		// State Change Condition
		IF (CIf.Job.bolAlmReset = FALSE) THEN
			IF (me.StateMachine.intStateHistory<=cSTA_PON) THEN
				me.StateMachine.intStateNext := cSTA_PONBusy;
			ELSIF (me.intCmd=cCMD_OFF) THEN
				me.StateMachine.intStateNext := cSTA_OFFBusy;
			ELSIF (me.intCmd=cCMD_RUN) THEN
				me.StateMachine.intStateNext := cSTA_OFFBusy;
			END_IF
		END_IF
	END_IF




//--------------------------------------------------------------------------------------
// Exit action
	IF (me.StateMachine.intState<>me.StateMachine.intStateNext) THEN
		;
	END_IF
END_METHOD

METHOD PROTECTED sta_OFF : BOOL
// state implemetation
//--------------------------------------------------------------------------------------
// Entry action
	IF (me.StateMachine.intState<>me.StateMachine.intStateLastCycle) THEN
		me.StateMachine.intStateLastCycle := me.StateMachine.intState;
		
	END_IF


//--------------------------------------------------------------------------------------
// Cyclic action
	IF (me.StateMachine.intState=me.StateMachine.intStateLastCycle) THEN
		
		;
		
		
		// State Change Condition
		IF (me.intCmd=cCMD_RUN) THEN
			me.StateMachine.intStateNext :=  cSTA_RUNBusy;
		END_IF
	END_IF




//--------------------------------------------------------------------------------------
// Exit action
	IF (me.StateMachine.intState<>me.StateMachine.intStateNext) THEN
		;
	END_IF
END_METHOD

METHOD PROTECTED sta_OFFBusy : BOOL
// state implemetation
//--------------------------------------------------------------------------------------
// Entry action
	IF (me.StateMachine.intState<>me.StateMachine.intStateLastCycle) THEN
		me.StateMachine.intStateLastCycle := me.StateMachine.intState;
		
	END_IF


//--------------------------------------------------------------------------------------
// Cyclic action
	IF (me.StateMachine.intState=me.StateMachine.intStateLastCycle) THEN
		pRFW_CIF^.Job.intACmd := cCMD_OFF;
		// send command OFF to all existing multi child controller. (Junctions)
		THIS^.CmdToAllMultiChild(cCMD_OFF);
	
		// State Change Condition
		IF (pRFW_CIF^.Job.intState = cSTA_OFF AND (THIS^.checkStateAllMultiChild(cSTA_OFF))) THEN
			me.StateMachine.intStateNext := cSTA_OFF;
		END_IF
	END_IF




//--------------------------------------------------------------------------------------
// Exit action
	IF (me.StateMachine.intState<>me.StateMachine.intStateNext) THEN
		;
	END_IF
END_METHOD

METHOD PROTECTED sta_PON : BOOL
// state implemetation
//--------------------------------------------------------------------------------------
// Entry action
	IF (me.StateMachine.intState<>me.StateMachine.intStateLastCycle) THEN
		me.StateMachine.intStateLastCycle := me.StateMachine.intState;
		
	END_IF


//--------------------------------------------------------------------------------------
// Cyclic action
	IF (me.StateMachine.intState=me.StateMachine.intStateLastCycle) THEN
		
		;
		
		
		// State Change Condition
		IF(me.intCmd=cCMD_OFF) OR (me.intCmd=cCMD_RUN) THEN
			me.StateMachine.intStateNext := cSTA_OFFBusy;
		END_IF
	END_IF




//--------------------------------------------------------------------------------------
// Exit action
	IF (me.StateMachine.intState<>me.StateMachine.intStateNext) THEN
		;
	END_IF
END_METHOD

METHOD PROTECTED sta_RUN : BOOL
// state implemetation
//--------------------------------------------------------------------------------------
// Entry action
	IF (me.StateMachine.intState<>me.StateMachine.intStateLastCycle) THEN
		me.StateMachine.intStateLastCycle := me.StateMachine.intState;

		uliRFID_Tag_old := pRFW_SIF^.Cur.stData.uliTagID; // Do no action with old datas

	END_IF


//--------------------------------------------------------------------------------------
// Cyclic action
	IF (me.StateMachine.intState=me.StateMachine.intStateLastCycle) THEN

		// Simulation
		IF (CIf.SwCfg.bolSimulation) THEN
			IF SIf.Cfg.bolSimSpeedInternal THEN
				SIf.Cur.dinTransportPosition_um := (SIf.Cur.dinTransportPosition_um + UDINT_TO_DINT(676 * me.FUBInfo.udiSample_ms)); // Speed TLPsort = 0.676 m/s = 676 um/ms
				SIf.Cur.dinTransportspeed_um_s := (676 * 1000);
			END_IF
			IF pRFW_SIF^.Cur.stData.uliTagID <> uliRFID_Tag_old THEN
				SIf.In.bolHangerDetector.intern := TRUE;
				dinPositionRFID_um := 0;
			ELSE
				SIf.In.bolHangerDetector.intern := FALSE;
			END_IF
		END_IF
		
		// Start the junctions if the output feeding is ok
		// Method send input command to all existing multi child controller.
		FOR intI:=0 TO usiNumOfMultiChild-1 BY 1 DO	
			IF SIf.Cur.a_bolJunctionOutputOK[intI] = TRUE THEN
				a_pMultiChildCIF[intI]^.Job.intACmd:= cCMD_RUN;
			ELSE
				a_pMultiChildCIF[intI]^.Job.intACmd:= cCMD_STOP;
			END_IF
		END_FOR


		// Increase the position of every Hanger in the hashtable, if it is on the way to junction
		dinTransportDifferenz_um := SIf.Cur.dinTransportPosition_um - dinTransportPosition_old_um;
		// Increase actual Position of the hanger at the RFID Reader Position if hanger there
		IF dinPositionRFID_um > 0 THEN
			dinPositionRFID_um := dinPositionRFID_um + dinTransportDifferenz_um;
		END_IF
		FOR uinLoopRFID := 0 TO INT_TO_UINT(cintMaxDecisions) DO
			IF aTblDecision[uinLoopRFID].dinActPos_um > 0 THEN
				aTblDecision[uinLoopRFID].dinActPos_um := aTblDecision[uinLoopRFID].dinActPos_um + dinTransportDifferenz_um;
			END_IF
		END_FOR	

		dinTransportPosition_old_um := SIf.Cur.dinTransportPosition_um;
			
	
		//--------------------------------------------------------------------------------------
		// Handle new RFID tags
		//--------------------------------------------------------------------------------------
		
		// RFID Reader gives a new Tag ID AND the sensor "Hanger detection" gives a Signal
		// Exactly position is from the sensor
		// But if sensor is first or the Tag ID is First is not defined!
		// If Sensor is first, write 1 into actual positon to increase
		// If RFID is first, write -1 To wait until sensor is detected
		
		// Check hanger detector sensor signal
		IF (SIf.In.bolHangerDetector.intern = TRUE) AND (bolREHangerDetection = FALSE) THEN
			bolREHangerDetection := TRUE;
			IF dinPositionRFID_um = 0 THEN //Sensor first
				dinPositionRFID_um := 1;
			ELSIF dinPositionRFID_um > 1 THEN	// Since last input no RFID Read
				// Set Alarm: SIf.Alm[5].strText := 'RFID Reader Tag not readed';
				pfbAlarmCtrl^.setAlarm(CIf.Info.intCtrlId,5,0,ADR(SIf.Alm),E_AlmState.RST,CIf.Job.eMe_ActivAlmClass);	
			ELSE	// RFID Tag Reader first
				aTblDecision[intIndexActualHanger].dinActPos_um := 1;
				dinPositionRFID_um := 0;
			END_IF
		ELSIF (SIf.In.bolHangerDetector.intern = FALSE) THEN
			bolREHangerDetection := FALSE;
		END_IF		
		
		
		// Check about new RFID Tag
		IF pRFW_SIF^.Cur.stData.uliTagID <> uliRFID_Tag_old THEN
			uliRFID_Tag_old := pRFW_SIF^.Cur.stData.uliTagID;
			bolJobFound := FALSE;
			// Loop through the hashtable to set new position
			FOR uinLoopRFID := 0 TO INT_TO_UINT(cintMaxDecisions) DO
				
				// Check if RFID already exists in buffer
				IF (aTblDecision[uinLoopRFID].stDecision.uliRFID = pRFW_SIF^.Cur.stData.uliTagID) THEN
					// Safe actual index for correct input
					intIndexActualHanger := UINT_TO_INT(uinLoopRFID);
					// Change state
					aTblDecision[uinLoopRFID].eState := E_DecisionState.WayToJunction;
					// Change timestamp
					aTblDecision[uinLoopRFID].dtTimeRFID := dtActualTime;
					
					// Check position, if RFID Reader first or Sensor first
					IF SIf.Cfg.bolHangerDetectionExist = FALSE THEN		// No exactly position detection
						dinPositionRFID_um := 0;
						// Start actual position with 1 to increase it cyclical
						aTblDecision[uinLoopRFID].dinActPos_um := dinPositionRFID_um;
					ELSIF dinPositionRFID_um = 0 THEN // RFID Reader first
						dinPositionRFID_um := -1;
					ELSIF dinPositionRFID_um = -1 THEN // Hanger detection does not detected a hanger
						// Set Alarm: SIf.Alm[6].strText := 'Hanger detection no hanger detected';
						pfbAlarmCtrl^.setAlarm(CIf.Info.intCtrlId,6,0,ADR(SIf.Alm),E_AlmState.RST,CIf.Job.eMe_ActivAlmClass);	
					ELSE	// Hanger detection first
						// Start actual position
						// ToDo: Tel. mit PRE. muss anders behandelt werden
						//aTblDecision[uinLoopRFID].dinActPos_um := dinPositionRFID_um;	
						aTblDecision[uinLoopRFID].dinActPos_um := 0;
						dinPositionRFID_um := -1;
					END_IF

					bolJobFound := TRUE;
					EXIT;
				END_IF
			END_FOR
			
			
			// RFID not exists in buffer. Create a new entry and set state to "WayToJunction". The target is not yet determined at this time.
			// Chance for line control to send a new job during the hanger is on the way to a junction.
			IF (bolJobFound = FALSE) THEN		
				// Search a free Element
				FOR uinLoopRFID := 0 TO INT_TO_UINT(cintMaxDecisions) DO
					
					// NO RFID = Free element
					IF (aTblDecision[uinLoopRFID].stDecision.uliRFID = 0) THEN					
						// Safe actual index for correct input
						intIndexActualHanger := UINT_TO_INT(uinLoopRFID);					
						// Save new RFID
						aTblDecision[uinLoopRFID].stDecision.uliRFID := pRFW_SIF^.Cur.stData.uliTagID;
						// Target=0, will be defined on the way to junction from line control
						aTblDecision[uinLoopRFID].stDecision.dinTarget := 0;				
						// Change state
						aTblDecision[uinLoopRFID].eState := E_DecisionState.WayToJunction;
						// Change timestamp
						aTblDecision[uinLoopRFID].dtTimeRFID := dtActualTime;
						
						// Check position, if RFID Reader first or Sensor first
						IF SIf.Cfg.bolHangerDetectionExist = FALSE THEN		// No exactly position detection
							dinPositionRFID_um := 0;
							// Start actual position with 1 to increase it cyclical
							aTblDecision[uinLoopRFID].dinActPos_um := dinPositionRFID_um;
						ELSIF dinPositionRFID_um = 0 THEN // RFID Reader first
							dinPositionRFID_um := -1;
						ELSIF dinPositionRFID_um = -1 THEN // Hanger detection does not detected a hanger
							// Set Alarm: SIf.Alm[6].strText := 'Hanger detection no hanger detected';
							pfbAlarmCtrl^.setAlarm(CIf.Info.intCtrlId,6,0,ADR(SIf.Alm),E_AlmState.RST,CIf.Job.eMe_ActivAlmClass);	 
						ELSE		// Hanger detection first
							// Start actual position
							// ToDo: Tel. mit PRE. muss anders behandelt werden
							//aTblDecision[uinLoopRFID].dinActPos_um := dinPositionRFID_um;	
							aTblDecision[uinLoopRFID].dinActPos_um := 0;
							dinPositionRFID_um := -1;										
						END_IF
							
						EXIT;
					END_IF
					
				END_FOR	
			END_IF
			
		END_IF		
		
		
		// State Change Condition
		// OFF done in always state
		IF (me.intCmd=cCMD_STOP) THEN
			me.StateMachine.intStateNext :=  cSTA_STOPBusy;	
		END_IF;
	END_IF




//--------------------------------------------------------------------------------------
// Exit action
	IF (me.StateMachine.intState<>me.StateMachine.intStateNext) THEN
		;
	END_IF
END_METHOD

METHOD PROTECTED sta_RUNBusy : BOOL
// state implemetation
//--------------------------------------------------------------------------------------
// Entry action
	IF (me.StateMachine.intState<>me.StateMachine.intStateLastCycle) THEN
		me.StateMachine.intStateLastCycle := me.StateMachine.intState;
		

		
		fbSimulationTimer.IN := FALSE;
		fbSimulationTimer.PT := UDINT_TO_TIME(SIf.Par.udiTimeOutRead_ms);
		fbSimulationTimer(); // set time/reset timer
		fbSimulationTimer.IN := TRUE; // start timer
	END_IF


//--------------------------------------------------------------------------------------
// Cyclic action
	IF (me.StateMachine.intState=me.StateMachine.intStateLastCycle) THEN

		// Simulation
		IF (CIf.SwCfg.bolSimulation) THEN
			fbSimulationTimer(); // simulation time
			IF (fbSimulationTimer.Q) THEN
				;
			END_IF
		END_IF
		
		// Cyclicle action
		pRFW_CIF^.Job.intACmd := cCMD_RUN;

		// State Change Condition
		IF (pRFW_CIF^.Job.intState = cSTA_RUN) THEN
			me.StateMachine.intStateNext := cSTA_RUN;
		ELSIF (me.intCmd=cCMD_STOP) THEN
			me.StateMachine.intStateNext :=  cSTA_STOPBusy;	
		END_IF
	END_IF




//--------------------------------------------------------------------------------------
// Exit action
	IF (me.StateMachine.intState<>me.StateMachine.intStateNext) THEN
		;
	END_IF
END_METHOD

METHOD PROTECTED sta_STOP : BOOL
// state implemetation
//--------------------------------------------------------------------------------------
// Entry action
	IF (me.StateMachine.intState<>me.StateMachine.intStateLastCycle) THEN
		me.StateMachine.intStateLastCycle := me.StateMachine.intState;

	END_IF


//--------------------------------------------------------------------------------------
// Cyclic action
	IF (me.StateMachine.intState=me.StateMachine.intStateLastCycle) THEN

		// Simulation
		IF (CIf.SwCfg.bolSimulation) THEN
			;
		END_IF
		
		// Increase the position of every Hanger in the hashtable, if it is on the way to junction
		dinTransportDifferenz_um := SIf.Cur.dinTransportPosition_um - dinTransportPosition_old_um;
		// Increase actual Position of the hanger at the RFID Reader Position if hanger there
		IF dinPositionRFID_um > 0 THEN
			dinPositionRFID_um := dinPositionRFID_um + dinTransportDifferenz_um;
		END_IF
		// Check in the same loop if any job is active
		bolNoJobActive := TRUE;
		FOR uinLoopRFID := 0 TO INT_TO_UINT(cintMaxDecisions) DO
			IF aTblDecision[uinLoopRFID].dinActPos_um > 0 THEN
				bolNoJobActive := FALSE;
				aTblDecision[uinLoopRFID].dinActPos_um := aTblDecision[uinLoopRFID].dinActPos_um + dinTransportDifferenz_um;
			END_IF
		END_FOR	

		dinTransportPosition_old_um := SIf.Cur.dinTransportPosition_um;
				
		IF (me.intCmd=cCMD_RUN) THEN
			me.StateMachine.intStateNext :=  cSTA_RUNBusy;	
		END_IF;
	END_IF




//--------------------------------------------------------------------------------------
// Exit action
	IF (me.StateMachine.intState<>me.StateMachine.intStateNext) THEN
		;
	END_IF
END_METHOD

METHOD PROTECTED sta_STOPBusy : BOOL
// state implemetation
//--------------------------------------------------------------------------------------
// Entry action
	IF (me.StateMachine.intState<>me.StateMachine.intStateLastCycle) THEN
		me.StateMachine.intStateLastCycle := me.StateMachine.intState;

	END_IF


//--------------------------------------------------------------------------------------
// Cyclic action
	IF (me.StateMachine.intState=me.StateMachine.intStateLastCycle) THEN

		// Simulation
		IF (CIf.SwCfg.bolSimulation) THEN
			IF SIf.Cfg.bolSimSpeedInternal THEN
				SIf.Cur.dinTransportPosition_um := (SIf.Cur.dinTransportPosition_um + UDINT_TO_DINT(676 * me.FUBInfo.udiSample_ms)); // Speed TLPsort = 0.676 m/s = 676 um/ms
				SIf.Cur.dinTransportspeed_um_s := (676 * 1000);
			END_IF
			IF pRFW_SIF^.Cur.stData.uliTagID <> uliRFID_Tag_old THEN
				SIf.In.bolHangerDetector.intern := TRUE;
				dinPositionRFID_um := 0;
			ELSE
				SIf.In.bolHangerDetector.intern := FALSE;
			END_IF
		END_IF
		
		// Increase the position of every Hanger in the hashtable, if it is on the way to junction
		dinTransportDifferenz_um := SIf.Cur.dinTransportPosition_um - dinTransportPosition_old_um;
		// Increase actual Position of the hanger at the RFID Reader Position if hanger there
		IF dinPositionRFID_um > 0 THEN
			dinPositionRFID_um := dinPositionRFID_um + dinTransportDifferenz_um;
		END_IF
		// Check in the same loop if any job is active
		bolNoJobActive := TRUE;
		FOR uinLoopRFID := 0 TO INT_TO_UINT(cintMaxDecisions) DO
(*			IF aTblDecision[uinLoopRFID].dinActPos_um > 0 THEN
				bolNoJobActive := FALSE;
				aTblDecision[uinLoopRFID].dinActPos_um := aTblDecision[uinLoopRFID].dinActPos_um + dinTransportDifferenz_um;
			END_IF
*)			IF ((aTblDecision[uinLoopRFID].eState = WayToJunction) OR (aTblDecision[uinLoopRFID].eState = OnJunction) OR
			(aTblDecision[uinLoopRFID].eState = Processed) OR (aTblDecision[uinLoopRFID].eState = DriveOut)) THEN
				bolNoJobActive := FALSE;
				aTblDecision[uinLoopRFID].dinActPos_um := aTblDecision[uinLoopRFID].dinActPos_um + dinTransportDifferenz_um;
			END_IF
		END_FOR	

		dinTransportPosition_old_um := SIf.Cur.dinTransportPosition_um;
				
		IF bolNoJobActive = TRUE THEN
			// send command OFF to all existing multi child controller. (Junctions)
			THIS^.CmdToAllMultiChild(cCMD_OFF);
		END_IF		
		
		
		// State Change Condition
		// OFF done in always state
		IF (THIS^.checkStateAllMultiChild(cSTA_OFF)) THEN
			me.StateMachine.intStateNext :=  cSTA_STOP;	
		ELSIF (me.intCmd=cCMD_RUN) THEN
			me.StateMachine.intStateNext :=  cSTA_RUNBusy;	
		END_IF;
	END_IF




//--------------------------------------------------------------------------------------
// Exit action
	IF (me.StateMachine.intState<>me.StateMachine.intStateNext) THEN
		;
	END_IF
END_METHOD

METHOD PROTECTED StateMachine : BOOL
SUPER^.StateMachine();

// main statemachine of base controller
CASE me.StateMachine.intState OF
    cSTA_RUNBusy: 
        THIS^.sta_RUNBusy();
    cSTA_RUN: 
        THIS^.sta_RUN();
    cSTA_STOPBusy: 
        THIS^.sta_STOPBusy();
    cSTA_STOP: 
        THIS^.sta_STOP();
END_CASE;
END_METHOD

END_FUNCTION_BLOCK

// POUs/Controller/Lvl1/DPJ (DecisionPoint Junction)/FB_DtChnToLine_JobDone
FUNCTION_BLOCK FB_DtChnToLine_JobDone
VAR_INPUT
	bolResetError: BOOL;
	pSIf: POINTER TO T_Ctrl_SIf_DPJ;
END_VAR
VAR_OUTPUT
	///Error value
	intError: INT;
END_VAR
VAR
	/// Internal Variable
	intStatemachine: INT;
	/// Data not correct
	bolDataBad: BOOL;
	/// Retry Counts for error message
	intCountRetry: INT;
	/// Buffer for Senddata
	aBuffer: ARRAY[0..cDtChnBuffer] OF T_JobDone_DtChn;
	/// Pointer for new Input
	intPBufferInput: INT;
	/// Pointer for readout
	intPBufferOutput: INT;
	/// Data Channel Specific Variable
	intIndexOldest: INT;
	/// Date and time of the oldes imput
	dtOldestTag: DT;
END_VAR
VAR CONSTANT
	cDtChnBuffer: INT := 20;
	cSTA_SUB_Data_Init: INT := 900;
	cSTA_SUB_Data_WaitForJob: INT := 902;
	cSTA_SUB_Data_SendData: INT := 904;
	cSTA_SUB_Data_Acknowledge: INT := 906;
	cSTA_SUB_Data_Retry: INT := 908;
	cSTA_SUB_Data_Error: INT := 910;
	cDataState_DONE: INT := -1;
	cDataState_Ready: INT := 1;
	cDataState_Retry: INT := -99;
	cDataState_Error: INT := -100;
	cMAX_RETRY: INT := 10;
	/// Error Codes
	cERR_NoSIF: INT := -100;
END_VAR

(*__________________________________________________________________________________________________
¦	
¦	Vistaprint Schweiz GmbH
¦	CH - 8401 Winterthur
¦
¦	www.vistaprint.ch - info@vistaprint.ch
¦___________________________________________________________________________________________________

Function desription:
Datachannel to send data to Lince Controller
Insert new Job with Method Creat in a Buffer
Send buffer elements if Linecontroller is ready


History:
Version		Date			Author		Comment
---------------------------------------------------------------------------------------------------
0.00.1		26.08.2013		AVM/PRE		Start history


___________________________________________________________________________________________________*)

// Data Channel to Receive Data from Line Controller
// Startup check States
IF (pSIf <> 0) THEN
	IF (intStatemachine < cSTA_SUB_Data_Init) THEN
		intStatemachine := cSTA_SUB_Data_Init;
	END_IF
ELSE
	intError := cERR_NoSIF;
END_IF

// 



CASE intStatemachine OF
	cSTA_SUB_Data_Init:
		IF pSIf^.DtChnToLine.stJobDone.intDataState = cDataState_DONE THEN
			intStatemachine := cSTA_SUB_Data_WaitForJob;
		END_IF
		
	cSTA_SUB_Data_WaitForJob:
		// New data arrived
		IF intPBufferInput <> intPBufferOutput THEN
			IF pSIf^.DtChnToLine.stJobDone.intDataState = cDataState_DONE THEN
				intStatemachine := cSTA_SUB_Data_SendData;
			END_IF
		END_IF
	
	cSTA_SUB_Data_SendData:	
		pSIf^.DtChnToLine.stJobDone.stDecision.uliRFID := aBuffer[intPBufferOutput].stDecision.uliRFID;
		pSIf^.DtChnToLine.stJobDone.stDecision.strID := aBuffer[intPBufferOutput].stDecision.strID;
		pSIf^.DtChnToLine.stJobDone.stDecision.dinTarget := aBuffer[intPBufferOutput].stDecision.dinTarget;
		pSIf^.DtChnToLine.stJobDone.strTimestamp := aBuffer[intPBufferOutput].strTimestamp;
		pSIf^.DtChnToLine.stJobDone.intDataState := cDataState_Ready;
		intStatemachine := cSTA_SUB_Data_Acknowledge;	
		
	cSTA_SUB_Data_Acknowledge:	
		IF pSIf^.DtChnToLine.stJobDone.intDataState = cDataState_DONE THEN
			// Data read from Line Controller
			// Reset Buffer Element
			aBuffer[intPBufferOutput].strTimestamp := '';
			aBuffer[intPBufferOutput].intDataState := 0;
			aBuffer[intPBufferOutput].stDecision.uliRFID := 0;
			aBuffer[intPBufferOutput].stDecision.strID := '';
			aBuffer[intPBufferOutput].stDecision.dinTarget := 0;
			// Increase Read out pointer
			IF intPBufferOutput < cDtChnBuffer THEN
				intPBufferOutput := intPBufferOutput + 1;
			ELSE
				intPBufferOutput := 0;
			END_IF
			intStatemachine := cSTA_SUB_Data_WaitForJob;
			
		ELSIF pSIf^.DtChnToLine.stJobDone.intDataState = cDataState_Retry THEN
			intStatemachine := cSTA_SUB_Data_Retry;
		ELSIF pSIf^.DtChnToLine.stJobDone.intDataState = cDataState_Error THEN
			intStatemachine := cSTA_SUB_Data_Error;
		END_IF
		
	cSTA_SUB_Data_Retry:
			IF intCountRetry < cMAX_RETRY THEN
				intCountRetry := intCountRetry + 1;
				intStatemachine := cSTA_SUB_Data_SendData;
			ELSE
				intStatemachine := cSTA_SUB_Data_Error;
			END_IF

	cSTA_SUB_Data_Error:
		intError := intCountRetry;
		IF bolResetError = TRUE THEN
			intStatemachine := cSTA_SUB_Data_WaitForJob;
		END_IF
			
END_CASE

METHOD Creat : INT
VAR_INPUT
	In_strTimestamp: STRING(24);
	In_stDecision: T_Decision;
END_VAR
// Insert a new Job to send at Line controller
// Only insert the job, if the buffer is not full, next input dosn't cross input and Outputpointer
IF ((intPBufferInput + 1) = intPBufferOutput) OR ((intPBufferInput = cDtChnBuffer) AND (intPBufferOutput = 0)) THEN
	Creat := -99;
ELSE
	aBuffer[intPBufferInput].stDecision.uliRFID := In_stDecision.uliRFID;
	aBuffer[intPBufferInput].stDecision.strID := In_stDecision.strID;
	aBuffer[intPBufferInput].stDecision.dinTarget := In_stDecision.dinTarget;
	aBuffer[intPBufferInput].strTimestamp := In_strTimestamp;
	IF intPBufferInput < cDtChnBuffer THEN
		intPBufferInput := intPBufferInput + 1;
	ELSE
		intPBufferInput := 0;
	END_IF
	Creat := 1;
END_IF
END_METHOD

END_FUNCTION_BLOCK

// POUs/Controller/Lvl2/COS (Control Station)/FB_COS
FUNCTION_BLOCK FB_COS EXTENDS FB_CtrlBase
VAR_INPUT
	/// push button next shirt
	In_bolNextShirt: BOOL;
	/// pointer to function block Slide Buffer
	p_fbSLB: POINTER TO FB_SLB;
	/// pointer to function block RFID
	p_fbRFW: POINTER TO FB_RFW;
	/// pointer to function block Single Stopper Buffer
	p_fbSSB: POINTER TO FB_STB;
	/// pointer to function block Drive
	p_fbTLS: POINTER TO FB_DRV;
END_VAR
VAR
	/// Specific interface struct for public access
	SIf: T_Ctrl_SIf_COS;
	/// Interface to Childs
	pSLB_CIF: POINTER TO T_Ctrl_CIf;
	pRFW_CIF: POINTER TO T_Ctrl_CIf;
	pSSB_CIF: POINTER TO T_Ctrl_CIf;
	pTLS_CIF: POINTER TO T_Ctrl_CIf;
	pSLB_SIF: POINTER TO T_Ctrl_SIf_SLB;
	pSSB_SIF: POINTER TO T_Ctrl_SIf_STB;
	/// Function specific variables
	/// edge detection push button
	usi_fpNextShirt: USINT;
END_VAR
VAR CONSTANT
	///sub States for RELEASE Function
	cSTA_SUB_WAIT_FOR_CMD: INT := 500;
	cSTA_SUB_SEND_RELEASE: INT := 501;
	cSTA_SUB_SEND_STOP: INT := 502;
END_VAR

(*__________________________________________________________________________________________________
¦	
¦	Vistaprint Schweiz GmbH
¦	CH - 8401 Winterthur
¦
¦	www.vistaprint.ch - info@vistaprint.ch
¦___________________________________________________________________________________________________

Function desription:
This module manages the flow of the shirts for checking the quality by the operator. 
As soon as the operator presses the button new shirt, the shirt at the operator stopper is released. 
After that the next shirt is released from the slide buffer to the operator stopper. 
The RFID readers communicate all the time the actual controlled shirt to the line controller. 
The ascending conveyor is running the whole time.

History:
Version		Date			Author		Comment
---------------------------------------------------------------------------------------------------
0.00.1		11.09.2013		AVM/KVO		Start history
0.00.2		04.12.2013		AVM/DSC		Input In_bolCounterIn, In_bolCounterOut and In_bolEmergencyOffOk deleted. 
										Handled in parent controller.
0.00.3		10.12.2013		AVM/DSC		Delete condition "me.Alarm.eActivAlmClass=E_AlmClass.STOP" in always method. 
										Don't change to state OFF_busy in case if active alm class is STOP.
0.00.4		16.12.2013		AVM/MRU		Overrule error always from base -> no EOFF State!! in EOFF go to OFF
						
___________________________________________________________________________________________________*)


IF ((me.bolActivate) AND (p_fbSLB<>0) AND (p_fbRFW<>0) AND (p_fbSSB<>0) AND (p_fbTLS<>0)) THEN // cyclic call enabled
	IF (CIf.Info.bolInitDone=FALSE) THEN // first cycle -> init
		CtrlInit();
		CIf.Info.bolInitDone := TRUE;
	ELSE
		CycleStartDuty();
	
		Always();
		
		StateMachine();
		
		CycleEndDuty();
	END_IF
END_IF;

METHOD PROTECTED Always : BOOL
IF (me.bolChangeBackToAUTO=TRUE) THEN // switch mode to automatic switch off controller
	//me.StateMachine.intStateNext := cSTA_OFFBusy;
	//me.bolChangeBackToAUTO := FALSE; // for cylinder no change to off when switch to automatic!!
END_IF

SUPER^.Always();

// ----------------------------------------------------------------------------------
// cyclic actions outside of statemachine
IF (me.StateMachine.intState<>cSTA_SINGLE_ANSWER) THEN
	;
END_IF


// ----------------------------------------------------------------------------------
// Always change actions in Base Library
// ----------------------------------------------------------------------------------
// overrule error always from base -> no EOFF State!! in EOFF go to OFF
IF (me.StateMachine.intStateNext = cSTA_EOFFBusy) THEN
	IF (me.StateMachine.intState=cSTA_OFF) THEN
		me.StateMachine.intStateNext := cSTA_OFF;
	ELSE // stay in OFF
		me.StateMachine.intStateNext := cSTA_OFFBusy;
	END_IF
END_IF

// Conditions Always
IF (((me.Alarm.eActivAlmClass=E_AlmClass.EOFF) OR (me.Alarm.eActivAlmClass=E_AlmClass.OFF) OR (me.intCmd=cCMD_OFF))
		 AND (me.StateMachine.intState<>cSTA_ERROR) AND (me.StateMachine.intState<>cSTA_ERRORQuit) AND
		(me.StateMachine.intState<>cSTA_OFF) AND (me.StateMachine.intState<>cSTA_OFFBusy)) THEN
	// alarm evt EOFF, OFF or cmd off
	me.StateMachine.intStateNext := cSTA_OFFBusy;
END_IF
END_METHOD

METHOD checkChildAlmClass : BOOL
//------------------------------------------------------------------------------------------------------
// check child alarm classes
IF (THIS^.CheckAllChildAlmClass(E_AlmClass.EOFF)) THEN
	CIf.Job.eMe_ActivAlmClass := E_AlmClass.EOFF;
	me.Alarm.bolfp := TRUE;
ELSIF (THIS^.CheckAllChildAlmClass(E_AlmClass.OFF)) THEN
	CIf.Job.eMe_ActivAlmClass := E_AlmClass.OFF;
	me.Alarm.bolfp := TRUE;
ELSIF (THIS^.CheckAllChildAlmClass(E_AlmClass.STOP)) THEN
	CIf.Job.eMe_ActivAlmClass := E_AlmClass.STOP;
	me.Alarm.bolfp := TRUE;
ELSE
	IF (me.Alarm.bolfp) THEN
		CIf.Job.eMe_ActivAlmClass := E_AlmClass.NONE; // no reset necessary
		me.Alarm.bolfp := FALSE;
	END_IF
END_IF

//------------------------------------------------------------------------------------------------------
// set alarm class parent of childs in the case of a parent EOFF or me=OFF or EOFF
IF (CIf.Job.eParent_ActivAlmClass=E_AlmClass.EOFF) THEN
	SetAllChildAlmClass(CIf.Job.eParent_ActivAlmClass);
ELSIF(CIf.Job.eMe_ActivAlmClass=E_AlmClass.EOFF) OR (CIf.Job.eMe_ActivAlmClass=E_AlmClass.OFF) THEN
	SetAllChildAlmClass(CIf.Job.eMe_ActivAlmClass);
ELSE
	// no important alarm for child active
	SetAllChildAlmClass(E_AlmClass.NONE);
END_IF
END_METHOD

METHOD PROTECTED CtrlInit : BOOL
VAR
	ii: INT;
	usiChildIndex: USINT;
END_VAR
SUPER^.CtrlInit();

pSLB_CIF := THIS^.AddChild(p_fbSLB^);
pRFW_CIF := THIS^.AddChild(p_fbRFW^);
pSSB_CIF := THIS^.AddChild(p_fbSSB^);
pTLS_CIF := THIS^.AddChild(p_fbTLS^);

// get specific interface for additional parmaeters or cur
pSLB_SIf := p_fbSLB^.getCtrlSIf();
pSSB_SIf := p_fbSSB^.getCtrlSIf();
//*******************************************************************************
// initial values childes
//*******************************************************************************
END_METHOD

METHOD FB_init : BOOL
VAR_INPUT
	///if TRUE, the retain variables are initialized (warm start / cold start)
	bInitRetains: BOOL;
	///if TRUE, the instance afterwards gets moved into the copy code (online change)
	bInCopyCode: BOOL;
END_VAR
VAR
	udiTaskCnt: UDINT;
	ii: UINT;
END_VAR
//------------------------------------------------------------------------------------------------------------------------
// to manually change in new FUB implementation!!!
// define valid commands for this controller
FOR ii:= 0 TO (SIZEOF(CIf.Job.aCmdList)/SIZEOF(CIf.Job.aCmdList[0])-1) BY 1 DO
	IF (CIf.Job.aCmdList[ii].intCmd=cCMD_INITIALIZED) THEN
		// found first empty array element
		EXIT;
	END_IF
END_FOR
CIf.Job.aCmdList[ii].intCmd := cCMD_RUN;
CIf.Job.aCmdList[ii].strName := 'Run'; 
CIf.Job.aCmdList[ii].bolAvailable := TRUE;
ii := ii +1;
CIf.Job.aCmdList[ii].intCmd := cCMD_STOP;
CIf.Job.aCmdList[ii].strName := 'Stop'; 
CIf.Job.aCmdList[ii].bolAvailable := TRUE;
ii := ii +1;

// set name of class/typ
CIf.Info.strType := 'FB_COS'; 

// set alarm class

//*******************************************************************************
// initial values
//*******************************************************************************

// software configuration
CIf.SwCfg.bolExist := TRUE;
CIf.SwCfg.bolSimulation := FALSE;

// Configuration

// parmeter
END_METHOD

METHOD PROTECTED getCmdState : STRING
VAR_INPUT
	intCmdState: INT;
	bolState: BOOL;
END_VAR
getCmdState := SUPER^.getCmdState(intCmdState:=intCmdState,bolState:=bolState); // get global/base defined cmds/states
IF (getCmdState='') THEN // global not defined get local
	// get string cmd/state string information in runtime
	IF (bolState=FALSE) THEN
		// cmd's
		CASE intCmdState OF
			COS_CmdState.cCMD_RELEASE:
				getCmdState := 'cCMD_RELEASE';
		END_CASE;
	ELSE
	
	// cmd's
		CASE intCmdState OF
			COS_CmdState.cSTA_RELEASEBusy:
				getCmdState := 'cSTA_RELEASEBusy';
			COS_CmdState.cSTA_RELEASE:
				getCmdState := 'cSTA_RELEASE';
				
			// SUB States
			cSTA_SUB_WAIT_FOR_CMD:
				getCmdState := 'cSTA_SUB_WAIT_FOR_CMD';
			cSTA_SUB_SEND_RELEASE:
				getCmdState := 'cSTA_SUB_SEND_RELEASE';
			cSTA_SUB_SEND_STOP:
				getCmdState := 'cSTA_SUB_SEND_STOP';
		END_CASE;
	END_IF
END_IF
END_METHOD

METHOD getCtrlSIf : POINTER TO T_Ctrl_SIf_COS
getCtrlSIf := ADR(SIf);
END_METHOD

METHOD PROTECTED IoInBridge : BOOL
// digitale and analoge inputs read from hardware or forcing
SIf.In.bolNextShirt.map := THIS^.In_bolNextShirt;

IF (CIf.SwCfg.bolSimulation = FALSE) THEN
	getInBol(CIf.Job.bolIoForce,ADR(SIf.In.bolNextShirt));
ELSE
	//simulation of global IO
END_IF
END_METHOD

METHOD PROTECTED sta_OFF : BOOL
// state implemetation
//--------------------------------------------------------------------------------------
// Entry action
	IF (me.StateMachine.intState<>me.StateMachine.intStateLastCycle) THEN
		me.StateMachine.intStateLastCycle := me.StateMachine.intState;

	END_IF


//--------------------------------------------------------------------------------------
// Cyclic action
	IF (me.StateMachine.intState=me.StateMachine.intStateLastCycle) THEN

		// Simulation
		IF (CIf.SwCfg.bolSimulation) THEN
			;
		END_IF
		
		// State Change Condition
		IF ((me.Alarm.eActivAlmClass<>E_AlmClass.EOFF) AND (me.Alarm.eActivAlmClass<>E_AlmClass.OFF)) THEN
			// enable start - no important error active
			IF(me.intCmd=cCMD_RUN) THEN
				me.StateMachine.intStateNext := cSTA_RUNBusy;
			END_IF
		END_IF
	END_IF




//--------------------------------------------------------------------------------------
// Exit action
	IF (me.StateMachine.intState<>me.StateMachine.intStateNext) THEN
		;
	END_IF
END_METHOD

METHOD PROTECTED sta_RUN : BOOL
// state implemetation
//--------------------------------------------------------------------------------------
// Entry action
	IF (me.StateMachine.intState<>me.StateMachine.intStateLastCycle) THEN
		me.StateMachine.intStateLastCycle := me.StateMachine.intState;
		
		me.SubStateMachine.intState := cSTA_SUB_WAIT_FOR_CMD; // init sub state machine
		me.SubStateMachine.intStateNext := cSTA_SUB_WAIT_FOR_CMD; // init sub state machine

	END_IF


//--------------------------------------------------------------------------------------
// Cyclic action
	IF (me.StateMachine.intState=me.StateMachine.intStateLastCycle) THEN

		// Simulation
		IF (CIf.SwCfg.bolSimulation) THEN
			;
		END_IF

		// positive edge detect -> release next shirt
		IF (SIf.In.bolNextShirt.intern=1) THEN
			IF (usi_fpNextShirt=0) THEN 
				usi_fpNextShirt := 1;
			END_IF
		ELSE
			usi_fpNextShirt := 0;
		END_IF
		
		CASE me.SubStateMachine.intState OF	
		// Start Cycle with substates	
		//--------------------------------------------------------------------------------------
		// sub state machine for sequence
		cSTA_SUB_WAIT_FOR_CMD:
		
			// Wait for command next shirt
			IF (usi_fpNextShirt=1) THEN
				usi_fpNextShirt := 2;
				me.SubStateMachine.intStateNext := cSTA_SUB_SEND_RELEASE;		
			ELSIF (me.intCmd=STB_CmdState.cCMD_RELEASE) THEN
				CIf.Job.intACmd:=cSTA_DONE;
				me.SubStateMachine.intStateNext := cSTA_SUB_SEND_RELEASE;		
			END_IF	
			
		cSTA_SUB_SEND_RELEASE:				
			// Send release command to single stopper
			pSSB_CIF^.Job.intACmd:= STB_CmdState.cCMD_RELEASE;

			// State Change Condition
			IF(pSSB_CIF^.Job.intState = STB_CmdState.cSTA_RELEASE)THEN
				me.SubStateMachine.intStateNext := cSTA_SUB_SEND_STOP;	
				pSLB_CIF^.Job.intACmd:= SLB_CmdState.cCMD_RELEASE;				
			END_IF		

		cSTA_SUB_SEND_STOP:
			// Send stop command to single stopper
			pSSB_CIF^.Job.intACmd:= cCMD_STOP;	
			
			// State Change Condition
			IF (pSSB_CIF^.Job.intState = cSTA_STOP) AND (CIf.Job.intACmd = cSTA_DONE)THEN
				me.SubStateMachine.intStateNext := cSTA_SUB_WAIT_FOR_CMD;																
			END_IF

		END_CASE
		
		me.SubStateMachine.intStateLastCycle := me.SubStateMachine.intState;
		CIf.Job.strSubState := THIS^.getCmdState(intCmdState:=me.SubStateMachine.intState,bolState:=TRUE);
		IF (me.SubStateMachine.intState<>me.SubStateMachine.intStateNext) THEN
			me.SubStateMachine.intState := me.SubStateMachine.intStateNext;  // set next state for next cycle
			me.SubStateMachine.udiTimeInState_ms := 0; // reset timer
			// log state change -> open point
		ELSE
			// increment time in state	
			me.SubStateMachine.udiTimeInState_ms := me.SubStateMachine.udiTimeInState_ms + me.FUBInfo.udiSample_ms;
		END_IF
				
		// State Change Condition	
		IF (me.intCmd=cCMD_STOP) THEN
			me.StateMachine.intStateNext :=  cSTA_STOPBusy;	
		END_IF
	END_IF

//--------------------------------------------------------------------------------------
// Exit action
	IF (me.StateMachine.intState<>me.StateMachine.intStateNext) THEN
		;
	END_IF
END_METHOD

METHOD PROTECTED sta_RUNBusy : BOOL
// state implemetation
//--------------------------------------------------------------------------------------
// Entry action
	IF (me.StateMachine.intState<>me.StateMachine.intStateLastCycle) THEN
		me.StateMachine.intStateLastCycle := me.StateMachine.intState;
		
	END_IF


//--------------------------------------------------------------------------------------
// Cyclic action
	IF (me.StateMachine.intState=me.StateMachine.intStateLastCycle) THEN

		// Simulation
		
		// Cyclic action
		pSLB_CIF^.Job.intACmd := cCMD_RUN;
		pRFW_CIF^.Job.intACmd := cCMD_RUN;
		
		IF ( (pSLB_CIF^.Job.intState = cSTA_RUN) AND (pRFW_CIF^.Job.intState = cSTA_RUN))  THEN
			pTLS_CIF^.Job.intACmd := cCMD_RUN;
			pSSB_CIF^.Job.intACmd := cCMD_STOP;
		END_IF;

		// State Change Condition
		IF ( (pSLB_CIF^.Job.intState = cSTA_RUN) AND (pRFW_CIF^.Job.intState = cSTA_RUN) AND
			(pSSB_CIF^.Job.intState = cSTA_STOP) AND (pTLS_CIF^.Job.intState = cSTA_RUN))  THEN
			me.StateMachine.intStateNext := cSTA_RUN;
		ELSIF (me.intCmd=cCMD_STOP) THEN
			me.StateMachine.intStateNext :=  cSTA_STOPBusy;	
		END_IF
	END_IF




//--------------------------------------------------------------------------------------
// Exit action
	IF (me.StateMachine.intState<>me.StateMachine.intStateNext) THEN
		;
	END_IF
END_METHOD

METHOD PROTECTED sta_STOP : BOOL
// state implemetation
//--------------------------------------------------------------------------------------
// Entry action
	IF (me.StateMachine.intState<>me.StateMachine.intStateLastCycle) THEN
		me.StateMachine.intStateLastCycle := me.StateMachine.intState;
		
	END_IF


//--------------------------------------------------------------------------------------
// Cyclic action
	IF (me.StateMachine.intState=me.StateMachine.intStateLastCycle) THEN
		
		;
		
		
		// State Change Condition
		IF (me.intCmd=cCMD_RUN) THEN
			me.StateMachine.intStateNext :=  cSTA_RUNBusy;
		END_IF
	END_IF




//--------------------------------------------------------------------------------------
// Exit action
	IF (me.StateMachine.intState<>me.StateMachine.intStateNext) THEN
		;
	END_IF
END_METHOD

METHOD PROTECTED sta_STOPBusy : BOOL
// state implemetation
//--------------------------------------------------------------------------------------
// Entry action
	IF (me.StateMachine.intState<>me.StateMachine.intStateLastCycle) THEN
		me.StateMachine.intStateLastCycle := me.StateMachine.intState;
		

	END_IF


//--------------------------------------------------------------------------------------
// Cyclic action
	IF (me.StateMachine.intState=me.StateMachine.intStateLastCycle) THEN

		// Simulation
		IF (CIf.SwCfg.bolSimulation) THEN
			;
		END_IF
		
		// Cyclicle action
		pSLB_CIF^.Job.intACmd := cCMD_STOP;

		IF (pSLB_CIF^.Job.intState = cCMD_STOP)  THEN
			pTLS_CIF^.Job.intACmd := cCMD_OFF;
			pSSB_CIF^.Job.intACmd := cCMD_STOP;
		END_IF;

		// State Change Condition
		IF ( (pSLB_CIF^.Job.intState = cSTA_STOP) AND (pSSB_CIF^.Job.intState = cSTA_STOP) AND (pTLS_CIF^.Job.intState = cSTA_OFF))  THEN
			me.StateMachine.intStateNext := cSTA_STOP;
		ELSIF (me.intCmd=cCMD_RUN) THEN
			me.StateMachine.intStateNext :=  cSTA_RUNBusy;	
		END_IF
	END_IF




//--------------------------------------------------------------------------------------
// Exit action
	IF (me.StateMachine.intState<>me.StateMachine.intStateNext) THEN
		;
	END_IF
END_METHOD

METHOD PROTECTED StateMachine : BOOL
SUPER^.StateMachine();

// main statemachine of base controller
CASE me.StateMachine.intState OF
    cSTA_RUNBusy: 
        THIS^.sta_RUNBusy();
    cSTA_RUN: 
        THIS^.sta_RUN();
    cSTA_STOPBusy: 
        THIS^.sta_STOPBusy();
    cSTA_STOP: 
        THIS^.sta_STOP();		
END_CASE;
END_METHOD

END_FUNCTION_BLOCK

// POUs/Controller/Lvl2/FOL (Folder)/FB_FOL
FUNCTION_BLOCK FB_FOL EXTENDS FB_CtrlBase
VAR_INPUT
	p_fbSLB: POINTER TO FB_SLB;
	/// CAN communication to folder
	p_fbFOC: POINTER TO FB_FOC;
	p_fbRFW: POINTER TO FB_RFW;
	p_fbTLS: POINTER TO FB_DRV;
END_VAR
VAR
	/// Specific interface struct for public access
	SIf: T_Ctrl_SIf_FOL;
	/// Child controller
	pSLB_CIf: POINTER TO T_Ctrl_CIf;
	/// CAN communication to folder
	pFOC_CIf: POINTER TO T_Ctrl_CIf;
	pRFW_CIf: POINTER TO T_Ctrl_CIf;
	pTLS_CIf: POINTER TO T_Ctrl_CIf;
	pSLB_SIF: POINTER TO T_Ctrl_SIf_SLB;
END_VAR
VAR CONSTANT
	cSTA_SUB_INITIALIZED: INT := 500;
	cSTA_SUB_START_ELEMENTS: INT := 502;
	cSTA_SUB_START_CYCLE: INT := 504;
	cSTA_SUB_START_WAIT_CYCLE: INT := 506;
	cSTA_SUB_START_FINAL: INT := 511;
	cSTA_SUB_FINISHED: INT := 600;
END_VAR

(*__________________________________________________________________________________________________
¦	
¦	Vistaprint Schweiz GmbH
¦	CH - 8401 Winterthur
¦
¦	www.vistaprint.ch - info@vistaprint.ch
¦___________________________________________________________________________________________________

Function desription:
Folder module instance controls Folder robot, slide buffer before folder, TLS conveyor for empty hangers and RFID reader in Folder.


History:
Version		Date			Author		Comment
---------------------------------------------------------------------------------------------------
0.00.1		01.10.2013		VP/RE		Start history
0.00.2		11.12.2013		AVME/MRU	Add Methode checkChildAlmClass for Error Stop of childs

___________________________________________________________________________________________________*)


// check if child pointer valid
IF ((me.bolActivate) AND (p_fbSLB<>0) AND (p_fbRFW<>0) AND (p_fbTLS<>0)) THEN // cyclic call enabled
	
	IF (CIf.Info.bolInitDone=FALSE) THEN // first cycle -> init
		CtrlInit();
		CIf.Info.bolInitDone := TRUE;
	ELSE
		CycleStartDuty();
	
		Always();
		
		StateMachine();
		
		CycleEndDuty();
	END_IF
	
END_IF;

METHOD PROTECTED Always : BOOL
IF (me.bolChangeBackToAUTO=TRUE) THEN // switch mode to automatic switch off controller
	//me.StateMachine.intStateNext := cSTA_OFFBusy;
	//me.bolChangeBackToAUTO := FALSE; // for cylinder no change to off when switch to automatic!!
END_IF

SUPER^.Always();

// ----------------------------------------------------------------------------------
// cyclic actions outside of statemachine
IF (me.StateMachine.intState<>cSTA_SINGLE_ANSWER) THEN
	;
END_IF

SIf.Cur.dinMaxCapacity := p_fbSLB^.getCtrlSIf()^.Cur.dinMaxCapacity;
SIf.Cur.bolIsFull := p_fbSLB^.getCtrlSIf()^.Cur.bolInputBufferFull;

// ----------------------------------------------------------------------------------
// Conditions Always
// overrule error always from base -> no EOFF State!! in EOFF go to OFF
IF (me.StateMachine.intStateNext = cSTA_EOFFBusy) THEN
	IF (me.StateMachine.intState=cSTA_OFF) THEN
		me.StateMachine.intStateNext := cSTA_OFF;
	ELSE // stay in OFF
		me.StateMachine.intStateNext := cSTA_OFFBusy;
	END_IF
END_IF
END_METHOD

METHOD checkChildAlmClass : BOOL
//------------------------------------------------------------------------------------------------------
// check child alarm classes
// set me alarm class active if at least one child has an EOFF
IF CheckAllChildAlmClass(E_AlmClass.EOFF) THEN
	CIf.Job.eMe_ActivAlmClass := E_AlmClass.EOFF;
	me.Alarm.bolfp := TRUE;
ELSIF CheckAllChildAlmClass(E_AlmClass.OFF) THEN
	CIf.Job.eMe_ActivAlmClass := E_AlmClass.OFF;
	me.Alarm.bolfp := TRUE;
ELSIF CheckAllChildAlmClass(E_AlmClass.STOP) THEN  // FB_MER needs alarm class STOP
	CIf.Job.eMe_ActivAlmClass := E_AlmClass.STOP;
	me.Alarm.bolfp := TRUE;
ELSE
	IF (me.Alarm.bolfp) THEN
		CIf.Job.eMe_ActivAlmClass := E_AlmClass.NONE; // no reset necessary
		me.Alarm.bolfp := FALSE;
	END_IF
END_IF

//------------------------------------------------------------------------------------------------------
// set alarm class parent of childs
//------------------------------------------------------------------------------------------------------
// set alarm class parent of childs in the case of a parent EOFF or me=OFF or EOFF
IF (CIf.Job.eParent_ActivAlmClass=E_AlmClass.EOFF) THEN
	SetAllChildAlmClass(CIf.Job.eParent_ActivAlmClass);
ELSIF(CIf.Job.eMe_ActivAlmClass=E_AlmClass.EOFF) OR (CIf.Job.eMe_ActivAlmClass=E_AlmClass.OFF) THEN
	SetAllChildAlmClass(CIf.Job.eMe_ActivAlmClass);
ELSE
	// no important alarm for child active
	SetAllChildAlmClass(E_AlmClass.NONE);
END_IF
END_METHOD

METHOD PROTECTED CtrlInit : BOOL
SUPER^.CtrlInit();

// get child CIf
pSLB_CIf := THIS^.AddChild(p_fbSLB^);
pFOC_CIf := THIS^.AddChild(p_fbFOC^);
pRFW_CIf := THIS^.AddChild(p_fbRFW^);
pTLS_CIf := THIS^.AddChild(p_fbTLS^);

pSLB_SIF := p_fbSLB^.getCtrlSIf();
END_METHOD

METHOD FB_init : BOOL
VAR_INPUT
	///if TRUE, the retain variables are initialized (warm start / cold start)
	bInitRetains: BOOL;
	///if TRUE, the instance afterwards gets moved into the copy code (online change)
	bInCopyCode: BOOL;
END_VAR
VAR
	ii: UINT;
END_VAR
//------------------------------------------------------------------------------------------------------------------------
// to manually change in new FUB implementation!!!
// define valid commands for this controller
FOR ii:= 0 TO (SIZEOF(CIf.Job.aCmdList)/SIZEOF(CIf.Job.aCmdList[0])-1) BY 1 DO
	IF (CIf.Job.aCmdList[ii].intCmd=cCMD_INITIALIZED) THEN
		// found first empty array element
		EXIT;
	END_IF
END_FOR
CIf.Job.aCmdList[ii].intCmd := cCMD_RUN;
CIf.Job.aCmdList[ii].strName := 'Run'; 
CIf.Job.aCmdList[ii].bolAvailable := TRUE;
//ii := ii +1;
//CIf.Job.aCmdList[ii].intCmd := cCMD_RETRACT;
//CIf.Job.aCmdList[ii].strName := 'Retract';
//CIf.Job.aCmdList[ii].bolAvailable := TRUE;

// set name of class/typ
CIf.Info.strType := 'FB_FOL'; 

// set alarm class
SIf.Alm[1].eAlmClass := E_AlmClass.INFO;
SIf.Alm[1].strText := 'Reserve'; 

//*******************************************************************************
// initial values
//*******************************************************************************

// software configuration
CIf.SwCfg.bolExist := TRUE;
CIf.SwCfg.bolSimulation := FALSE;

// parmeter
//SIf.Par.udiDelayFirstClamp_ms := 750;

// actual values
//SIf.Cur.dinCounter := 0;
END_METHOD

METHOD PROTECTED getCmdState : STRING
VAR_INPUT
	intCmdState: INT;
	bolState: BOOL;
END_VAR
getCmdState := SUPER^.getCmdState(intCmdState:=intCmdState,bolState:=bolState); // get global/base defined cmds/states

IF (getCmdState='') THEN // global not defined get local
	// get string cmd/state string information in runtime
	IF (bolState=FALSE) THEN
		// cmd's
	ELSE
	
	// cmd's
		CASE intCmdState OF
				
			// SUB States
			cSTA_SUB_INITIALIZED:
				getCmdState := 'cSTA_SUB_INITIALIZED';
			cSTA_SUB_START_CYCLE:
				getCmdState := 'cSTA_SUB_START_CYCLE';
			cSTA_SUB_START_Wait_CYCLE:
				getCmdState := 'cSTA_SUB_START_Wait_CYCLE';
			cSTA_SUB_START_ELEMENTS:
				getCmdState := 'cSTA_SUB_START_ELEMENTS';
			cSTA_SUB_START_FINAL:
				getCmdState := 'cSTA_SUB_START_FINAL';
			cSTA_SUB_FINISHED:
				getCmdState := 'cSTA_SUB_FINISHED';
		END_CASE;
	END_IF
END_IF
END_METHOD

METHOD getCtrlSIf : POINTER TO T_Ctrl_SIf_FOL
getCtrlSIf := ADR(SIf);
END_METHOD

METHOD PROTECTED IoInBridge : BOOL
// digitale and analoge inputs read from hardware or forcing
//SIf.In.bolEmergencyStop.map := THIS^.In_EmergencyStop;

IF (CIf.SwCfg.bolSimulation = FALSE) THEN
	//getInBol(CIf.Job.bolIoForce,ADR(SIf.In.bolEmergencyStop));
ELSE
	//simulation of global IO
END_IF
END_METHOD

METHOD PROTECTED IoOutBridge : BOOL
VAR
	bolSwitchValvesOff: BOOL;
END_VAR
// digitale and analoge inputs read from hardware or forcing
IF (CIf.SwCfg.bolSimulation = FALSE) THEN
//	setOutBol(CIf.Job.bolIoForce ,ADR(SIf.Out.bolClamping));

//	THIS^.Out_Clamping := SIf.Out.bolClamping.map;
END_IF
END_METHOD

METHOD PROTECTED sta_OFF : BOOL
// state implemetation
//--------------------------------------------------------------------------------------
// Entry action
	IF (me.StateMachine.intState<>me.StateMachine.intStateLastCycle) THEN
		me.StateMachine.intStateLastCycle := me.StateMachine.intState;
		
	END_IF

//--------------------------------------------------------------------------------------
// Cyclic action
	IF (me.StateMachine.intState=me.StateMachine.intStateLastCycle) THEN
				
		// State Change Condition
		IF ((me.Alarm.eActivAlmClass<>E_AlmClass.EOFF) AND (me.Alarm.eActivAlmClass<>E_AlmClass.OFF)) THEN
			// enable start - no important error active
			IF me.intCmd=cCMD_RUN THEN
				me.StateMachine.intStateNext :=  cSTA_RUNBusy;
			END_IF
		END_IF
	END_IF


//--------------------------------------------------------------------------------------
// Exit action
	IF (me.StateMachine.intState<>me.StateMachine.intStateNext) THEN
		;
	END_IF
END_METHOD

METHOD PROTECTED sta_RUN : BOOL
// state implemetation
//--------------------------------------------------------------------------------------
// Entry action
	IF (me.StateMachine.intState<>me.StateMachine.intStateLastCycle) THEN
		me.StateMachine.intStateLastCycle := me.StateMachine.intState;
	
		me.SubStateMachine.intState := cSTA_SUB_START_CYCLE; // init sub state machine
		me.SubStateMachine.intStateNext := cSTA_SUB_START_CYCLE; // init sub state machine		
	END_IF

//--------------------------------------------------------------------------------------
// Cyclic action
	IF (me.StateMachine.intState=me.StateMachine.intStateLastCycle) THEN

		// Simulation
		IF (CIf.SwCfg.bolSimulation) THEN
			;
		END_IF

		// sub state machine for sequence
		CASE me.SubStateMachine.intState OF

			cSTA_SUB_START_CYCLE:	
				IF (pSLB_SIF^.Cur.bolHangerDetected) THEN
					pSLB_CIf^.Job.intACmd := SLB_CmdState.cCMD_RELEASE;
					me.SubStateMachine.intStateNext := cSTA_SUB_FINISHED;
				END_IF
			
			cSTA_SUB_FINISHED:	
				// Wait until job done
				IF(pSLB_CIf^.Job.intACmd = cSTA_DONE)THEN	
					IF (me.SubStateMachine.udiTimeInState_ms >= SIf.Par.udiTimeNextHangers_ms) THEN
						me.SubStateMachine.intStateNext := cSTA_SUB_START_CYCLE;
					END_IF
				END_IF	
		END_CASE

		// State Change Condition	
		IF (me.intCmd=BASE_PLC.cCMD_OFF) THEN
			me.StateMachine.intStateNext :=  cSTA_OFFBusy;	
		END_IF
	END_IF

//--------------------------------------------------------------------------------------
// Exit action
	IF (me.StateMachine.intState<>me.StateMachine.intStateNext) THEN
		;
	END_IF
END_METHOD

METHOD PROTECTED sta_RUNBusy : BOOL
// state implemetation
//--------------------------------------------------------------------------------------
// Entry action
	IF (me.StateMachine.intState<>me.StateMachine.intStateLastCycle) THEN
		me.StateMachine.intStateLastCycle := me.StateMachine.intState;
		
		me.SubStateMachine.intState := cSTA_SUB_INITIALIZED; // init sub state machine
		me.SubStateMachine.intStateNext := cSTA_SUB_INITIALIZED; // init sub state machine
	END_IF

//--------------------------------------------------------------------------------------
// Cyclic action
	IF (me.StateMachine.intState=me.StateMachine.intStateLastCycle) THEN

		// Simulation
		IF (CIf.SwCfg.bolSimulation) THEN
			fbSimulationTimer(); // simulation time
			IF (fbSimulationTimer.Q) THEN
				;
			END_IF
		END_IF
		
		// Cyclicle action
		// Start Cycle with substates	
		//--------------------------------------------------------------------------------------
		// sub state machine for sequence
		CASE me.SubStateMachine.intState OF
			//--------------------------------------------------------------------------------------
			cSTA_SUB_INITIALIZED:
				me.SubStateMachine.intStateNext := cSTA_SUB_START_ELEMENTS;
				
			cSTA_SUB_START_ELEMENTS:
				//start all childs
				pSLB_CIf^.Job.intACmd := cCMD_RUN;
				pFOC_CIf^.Job.intACmd := cCMD_RUN;
				pRFW_CIf^.Job.intACmd := cCMD_RUN;
				pTLS_CIf^.Job.intACmd := cCMD_RUN;
	
				IF ((pSLB_CIf^.Job.intState = cSTA_RUN) AND (pRFW_CIf^.Job.intState = cSTA_RUN) AND (pTLS_CIf^.Job.intState = cSTA_RUN) AND (pFOC_CIf^.Job.intState = cSTA_RUN)) THEN
					me.SubStateMachine.intStateNext := cSTA_SUB_FINISHED;
				END_IF
				
		//--------------------------------------------------------------------------------------
			cSTA_SUB_FINISHED:
					;
					
		END_CASE
			
		// State Change Condition
		IF (me.SubStateMachine.intState = cSTA_SUB_FINISHED) THEN
			me.StateMachine.intStateNext := cSTA_RUN;
		ELSIF (me.intCmd=cCMD_STOP) THEN
			me.StateMachine.intStateNext :=  cSTA_STOPBusy;	
		END_IF
	END_IF

//--------------------------------------------------------------------------------------
// Exit action
	IF (me.StateMachine.intState<>me.StateMachine.intStateNext) THEN
		;
	END_IF
END_METHOD

METHOD PROTECTED StateMachine : BOOL
SUPER^.StateMachine();

// main statemachine of base controller
CASE me.StateMachine.intState OF
    cSTA_RUNBusy: 
        THIS^.sta_RUNBusy();
    cSTA_RUN: 
        THIS^.sta_RUN();
END_CASE;
END_METHOD

END_FUNCTION_BLOCK

// POUs/Controller/Lvl2/HFE/FB_HFE
FUNCTION_BLOCK FB_HFE EXTENDS FB_CtrlBase
VAR_INPUT
	a_bolLDSNeedsHanger: ARRAY[0..cuintMaxStation] OF BOOL;
	a_intHFE_BufferZone: ARRAY[0..cuintMaxStation] OF INT;
	p_fbTlpDrive: POINTER TO FB_DRV;
	///p_fbJunction : POINTER TO FB_JUN;
	p_fbSLB: POINTER TO FB_SLB;
END_VAR
VAR
	/// List of pointers to Childs of VLV
	a_pMultiChildCtrl: ARRAY[0..Base_Const.cMaxNrOfChilds] OF POINTER TO FB_VLV;
	/// List of childs common interface
	a_pMultiChildCIF: ARRAY[0..Base_Const.cMaxNrOfChilds] OF POINTER TO T_Ctrl_CIf;
	/// List of childs specific interface for additional parameters or cur
	a_pMultiChildSIF: ARRAY[0..Base_Const.cMaxNrOfChilds] OF POINTER TO Base_Elements.T_Ctrl_SIf_VLV;
	usiNumOfMultiChild: USINT;
	usiNumOfValidPointerMultiChild: USINT;
	/// Specific interface struct for public access
	SIf: T_Ctrl_SIf_HFE;
	/// Child controller
	pTlpDrive_CIf: POINTER TO T_Ctrl_CIf;
	///pJunction_CIf : POINTER TO T_Ctrl_CIf;
	pSLB_CIf: POINTER TO T_Ctrl_CIf;
	pSLB_SIf: POINTER TO T_Ctrl_SIf_SLB;
	intSubState: ARRAY[0..cuintMaxStation] OF INT;
	udiTimeInStateRefill_ms: ARRAY[0..cuintMaxStation] OF UDINT;
END_VAR
VAR CONSTANT
	/// sub States
	cSTA_SUB_WaitForJob: INT := 500;
	cSTA_SUB_WaitOpen: INT := 502;
	cSTA_SUB_Open: INT := 504;
	cSTA_SUB_WaitClose: INT := 506;
	cSTA_SUB_Close: INT := 508;
END_VAR

(*__________________________________________________________________________________________________
¦	
¦	Vistaprint Schweiz GmbH
¦	CH - 8401 Winterthur
¦
¦	www.vistaprint.ch - info@vistaprint.ch
¦___________________________________________________________________________________________________

Function desription:
Cylinder implementation. 


History:
Version		Date			Author		Comment
---------------------------------------------------------------------------------------------------
0.00.1		02.07.2013		VP/RE		Start history
0.00.2		16.12.2013		AVME/MRU	In Always: No EOFF State!! in EOFF go to OFF

___________________________________________________________________________________________________*)



// check if child pointer valid
IF (me.bolActivate) AND (p_fbTlpDrive<>0)  AND (THIS^.checkChildPointer()) AND (p_fbSLB<>0) THEN // cyclic call enabled
	
	IF (CIf.Info.bolInitDone=FALSE) THEN // first cycle -> init
		CtrlInit();
		CIf.Info.bolInitDone := TRUE;
	ELSE
		CycleStartDuty();
	
		Always();
		
		StateMachine();
		
		CycleEndDuty();
	END_IF
	
END_IF;

METHOD AddJunction
VAR_INPUT
	p_MultiChild: POINTER TO FB_JUN;
END_VAR

// Method add the pointer address of the buffer zone child controller to the array list.
IF (usiNumOfMultiChild <= (Base_Const.cMaxNrOfChilds-1)) THEN
	// Add buffer zone child controller to list
	a_pMultiChildCtrl[usiNumOfMultiChild] := p_MultiChild;
	// Inc. number of buffer zones
	usiNumOfMultiChild:= usiNumOfMultiChild+1;
	// Check if the pointer is valid
	IF (p_MultiChild<>0) THEN
		usiNumOfValidPointerMultiChild:= usiNumOfValidPointerMultiChild+1;
	END_IF
END_IF
END_METHOD

METHOD PROTECTED Always : BOOL
SUPER^.Always();

IF (me.StateMachine.intState<>cSTA_SINGLE_ANSWER) THEN
	
	;
	
END_IF

// ----------------------------------------------------------------------------------
// Conditions Always
// overrule error always from base -> no EOFF State!! in EOFF go to OFF
IF (me.StateMachine.intStateNext = cSTA_EOFFBusy) THEN
	IF (me.StateMachine.intState=cSTA_OFF) THEN
		me.StateMachine.intStateNext := cSTA_OFF;
	ELSE // stay in OFF
		me.StateMachine.intStateNext := cSTA_OFFBusy;
	END_IF
END_IF
END_METHOD

METHOD PROTECTED checkChildPointer : BOOL
IF (usiNumOfMultiChild = usiNumOfValidPointerMultiChild) THEN
	checkChildPointer:= TRUE;
ELSE
	checkChildPointer:= FALSE;
END_IF
END_METHOD

METHOD PROTECTED CtrlInit : BOOL
VAR
	ii: INT;
END_VAR
SUPER^.CtrlInit();

// get child CIf
pTlpDrive_CIf := THIS^.AddChild(p_fbTlpDrive^);
pSLB_CIf := THIS^.AddChild(p_fbSLB^);
pSLB_SIf := p_fbSLB^.getCtrlSIf();

//initialize all multi Child controller.
FOR ii:=0 TO usiNumOfMultiChild-1 BY 1 DO	
	// Get child common if
	a_pMultiChildCIF[ii]:= THIS^.AddChild(a_pMultiChildCtrl[ii]^);	
	// Get specific interface for additional parmaeters or cur
	a_pMultiChildSIF[ii]:= a_pMultiChildCtrl[ii]^.getCtrlSIf();
END_FOR
END_METHOD

METHOD FB_init : BOOL
VAR_INPUT
	///if TRUE, the retain variables are initialized (warm start / cold start)
	bInitRetains: BOOL;
	///if TRUE, the instance afterwards gets moved into the copy code (online change)
	bInCopyCode: BOOL;
END_VAR
VAR
	ii: UINT;
END_VAR
//------------------------------------------------------------------------------------------------------------------------
// to manually change in new FUB implementation!!!
// define valid commands for this controller
FOR ii:= 0 TO (SIZEOF(CIf.Job.aCmdList)/SIZEOF(CIf.Job.aCmdList[0])-1) BY 1 DO
	IF (CIf.Job.aCmdList[ii].intCmd=cCMD_INITIALIZED) THEN
		// found first empty array element
		EXIT;
	END_IF
END_FOR
CIf.Job.aCmdList[ii].intCmd := cCMD_RUN;
CIf.Job.aCmdList[ii].strName := 'Run'; 
CIf.Job.aCmdList[ii].bolAvailable := TRUE;
//ii := ii +1;
//CIf.Job.aCmdList[ii].intCmd := cCMD_RETRACT;
//CIf.Job.aCmdList[ii].strName := 'Retract';
//CIf.Job.aCmdList[ii].bolAvailable := TRUE;

// set name of class/typ
CIf.Info.strType := 'FB_HFE'; 

// set alarm class
//SIf.Alm[1].eAlmClass := E_AlmClass.TSTOP;
//SIf.Alm[1].strText := 'TLKV Motor does not move after timeout.'; 
//SIf.Alm[2].eAlmClass := E_AlmClass.STOP;
//SIf.Alm[2].strText := 'Emergency button pressed.'; 

//*******************************************************************************
// initial values
//*******************************************************************************

// software configuration
CIf.SwCfg.bolExist := TRUE;
CIf.SwCfg.bolSimulation := FALSE;

// parmeter
SIf.Par.udiWaitingTime_ms := 100;
SIf.Par.a_bolEnableJunction[0] := TRUE; // First LDS is enabled

// configuration
SIf.Cfg.uintNbOfLDS := 1;

// actual values
//SIf.Cur.dinCounter := 0;
END_METHOD

METHOD getCtrlSIf : POINTER TO T_Ctrl_SIf_HFE
getCtrlSIf := ADR(SIf);
END_METHOD

METHOD PROTECTED IoInBridge : BOOL
// digitale and analoge inputs read from hardware or forcing
//SIf.In.bolGiveNextHangerSensor.map := THIS^.In_GiveNextHangerSensor;

IF (CIf.SwCfg.bolSimulation = FALSE) THEN
	//getInBol(CIf.Job.bolIoForce,ADR(SIf.In.bolGiveNextHangerSensor));
ELSE
	//simulation of global IO
END_IF
END_METHOD

METHOD PROTECTED IoOutBridge : BOOL
VAR
	bolSwitchValvesOff: BOOL;
END_VAR
// digitale and analoge inputs read from hardware or forcing
IF (CIf.SwCfg.bolSimulation = FALSE) THEN
	//setOutBol(CIf.Job.bolIoForce ,ADR(SIf.Out.bolClamping));

	//THIS^.Out_Clamping := SIf.Out.bolClamping.map;
END_IF
END_METHOD

METHOD Refill
VAR_INPUT
	intNbOfLDS: INT;
END_VAR
VAR
	/// Loop variable
	ii: INT;
END_VAR
// Simulation
fbSimulationTimer.PT := UDINT_TO_TIME(1000);
IF (CIf.SwCfg.bolSimulation) THEN
	// Cyclicle input into the top stopperbuffer
	fbSimulationTimer(); // set time/reset timer
	IF fbSimulationTimer.Q = TRUE THEN
		fbSimulationTimer.IN := FALSE;
	ELSE
		fbSimulationTimer.IN := TRUE;
	END_IF
			
END_IF

// Method refill 
CASE intSubState[intNbOfLDS] OF
	cSTA_SUB_WaitForJob: // LDS needs hanger
		IF (a_bolLDSNeedsHanger[intNbOfLDS]) THEN
//			IF (p_fbSLB^.CtrlCIf^.Info.p_aCIf[intNbOfLDS + 2]^.job.intState = 6) OR (p_fbSLB^.CtrlCIf^.Info.p_aCIf[intNbOfLDS + 2]^.job.intState = 12) THEN //	Just open if PreStopper is closed
			IF (p_fbSLB^.CtrlCIf^.Info.p_aCIf[a_intHFE_BufferZone[intNbOfLDS]]^.job.intState = 6) 
			OR (p_fbSLB^.CtrlCIf^.Info.p_aCIf[a_intHFE_BufferZone[intNbOfLDS]]^.job.intState = 12) THEN //	Just open if PreStopper is closed
				a_pMultiChildCIF[intNbOfLDS]^.Job.intACmd:= Base_Elements.VLV_CmdState.cCMD_OPEN;
				udiTimeInStateRefill_ms[intNbOfLDS] := 0;
				intSubState[intNbOfLDS] := cSTA_SUB_WaitOpen;
			END_IF
		END_IF
	
	cSTA_SUB_WaitOpen:	// Waiting time between STB closing and junction opening
		udiTimeInStateRefill_ms[intNbOfLDS]:= udiTimeInStateRefill_ms[intNbOfLDS] + me.FUBInfo.udiSample_ms;
		IF (udiTimeInStateRefill_ms[intNbOfLDS] > SIf.Par.udiWaitingTime_ms) THEN
			intSubState[intNbOfLDS] := cSTA_SUB_Open;
		END_IF
		
	cSTA_SUB_Open:	
		IF (a_bolLDSNeedsHanger[intNbOfLDS] = 0) THEN
			intSubState[intNbOfLDS] := cSTA_SUB_WaitClose;
		END_IF
		
	cSTA_SUB_WaitClose:	// Waiting time between STB closing and junction closing
//		IF (p_fbSLB^.CtrlCIf^.Info.p_aCIf[intNbOfLDS + 2]^.job.intState = 6) or (p_fbSLB^.CtrlCIf^.Info.p_aCIf[intNbOfLDS + 2]^.job.intState = 12) THEN //	Just close if PreStopper is closed
		IF (p_fbSLB^.CtrlCIf^.Info.p_aCIf[a_intHFE_BufferZone[intNbOfLDS]]^.job.intState = 6) 
		OR (p_fbSLB^.CtrlCIf^.Info.p_aCIf[a_intHFE_BufferZone[intNbOfLDS]]^.job.intState = 12) THEN //	Just close if PreStopper is closed

			udiTimeInStateRefill_ms[intNbOfLDS] := 0;
			intSubState[intNbOfLDS] := cSTA_SUB_Close;
		END_IF
		
	cSTA_SUB_Close:
		udiTimeInStateRefill_ms[intNbOfLDS]:= udiTimeInStateRefill_ms[intNbOfLDS] + me.FUBInfo.udiSample_ms;
		IF (udiTimeInStateRefill_ms[intNbOfLDS] > SIf.Par.udiWaitingTime_ms) THEN
			a_pMultiChildCIF[intNbOfLDS]^.Job.intACmd:= Base_Elements.VLV_CmdState.cCMD_Close;
			intSubState[intNbOfLDS] := cSTA_SUB_WaitForJob;
		END_IF
END_CASE
END_METHOD

METHOD PROTECTED sta_OFF : BOOL
// state implemetation
//--------------------------------------------------------------------------------------
// Entry action
	IF (me.StateMachine.intState<>me.StateMachine.intStateLastCycle) THEN
		me.StateMachine.intStateLastCycle := me.StateMachine.intState;
		
	END_IF


//--------------------------------------------------------------------------------------
// Cyclic action
	IF (me.StateMachine.intState=me.StateMachine.intStateLastCycle) THEN
		
		;
		
		// State Change Condition
		IF me.intCmd=cCMD_RUN THEN
			me.StateMachine.intStateNext :=  cSTA_RUNBusy;
		END_IF
	END_IF




//--------------------------------------------------------------------------------------
// Exit action
	IF (me.StateMachine.intState<>me.StateMachine.intStateNext) THEN
		;
	END_IF
END_METHOD

METHOD PROTECTED sta_RUN : BOOL
VAR
	intNbOfLDS: INT;
END_VAR
// state implemetation
//--------------------------------------------------------------------------------------
// Entry action
	IF (me.StateMachine.intState<>me.StateMachine.intStateLastCycle) THEN
		me.StateMachine.intStateLastCycle := me.StateMachine.intState;
		
		//fbSimulationTimer.IN := FALSE;
		//fbSimulationTimer.PT := UDINT_TO_TIME(SIf.Par.udi_pulseTimeout_ms/10);
		//fbSimulationTimer(); // set time/reset timer
		//fbSimulationTimer.IN := TRUE; // start timer
		FOR intNbOfLDS := 0 TO cuintMaxStation DO
			intSubState[intNbOfLDS] := 500;	// Init Refill Substate
		END_FOR
	END_IF


//--------------------------------------------------------------------------------------
// Cyclic action
	IF (me.StateMachine.intState=me.StateMachine.intStateLastCycle) THEN
		
		// Simulation
		IF (CIf.SwCfg.bolSimulation) THEN
			//fbSimulationTimer(); // simulation time
			//IF (fbSimulationTimer.Q) THEN
			//	SIf.In.bolPulse.intern := NOT SIf.In.bolPulse.intern; // toggle pulse
			//	fbSimulationTimer.IN := FALSE;
			//ELSE
			//	fbSimulationTimer.IN := TRUE;
			//END_IF
		END_IF
		
		//IF NOT(pSLB_SIf^.Cur.bolBufferFull) THEN
		//	pStopperBuffer_CIf^.Job.intACmd := STB_CmdState.cCMD_RELEASE;
		//END_IF
		FOR intNbOfLDS := 0 TO cuintMaxStation DO
			IF (SIf.Par.a_bolEnableJunction[intNbOfLDS]) AND (a_pMultiChildCtrl[intNbOfLDS]<>0) THEN
				Refill(intNbOfLDS);
			END_IF
			IF (INT_TO_UINT(intNbOfLDS) = (SIf.Cfg.uintNbOfLDS-1)) THEN // Last station = End of SLB, no VLV there
				IF (a_bolLDSNeedsHanger[intNbOfLDS]= TRUE) THEN
					IF (pSLB_SIf^.Cur.bolHangerDetected = TRUE) THEN // Just if Hanger is at Last STB
						pSLB_CIf^.Job.intACmd := SLB_CmdState.cCMD_RELEASE;	
					END_IF
				END_IF
			END_IF
		END_FOR
		
		// State Change Condition
		IF me.intCmd=cCMD_OFF THEN
			me.StateMachine.intStateNext := cSTA_OFFBusy;
		END_IF
		
	END_IF



//--------------------------------------------------------------------------------------
// Exit action
	IF (me.StateMachine.intState<>me.StateMachine.intStateNext) THEN
		;
	END_IF
END_METHOD

METHOD PROTECTED sta_RUNBusy : BOOL
// state implemetation
//--------------------------------------------------------------------------------------
// Entry action
	IF (me.StateMachine.intState<>me.StateMachine.intStateLastCycle) THEN
		me.StateMachine.intStateLastCycle := me.StateMachine.intState;
		
		pTlpDrive_CIf^.Job.intACmd := cCMD_RUN;
		pSLB_CIf^.Job.intACmd := Base_PLC.cCMD_RUN;
		
	END_IF


//--------------------------------------------------------------------------------------
// Cyclic action
	IF (me.StateMachine.intState=me.StateMachine.intStateLastCycle) THEN
		
		// State Change Condition
		IF (pTlpDrive_CIf^.Job.intState = cSTA_RUN) THEN
			me.StateMachine.intStateNext := cSTA_RUN;
		END_IF
	END_IF



//--------------------------------------------------------------------------------------
// Exit action
	IF (me.StateMachine.intState<>me.StateMachine.intStateNext) THEN
		;
	END_IF
END_METHOD

METHOD PROTECTED StateMachine : BOOL
SUPER^.StateMachine();

// main statemachine of base controller
CASE me.StateMachine.intState OF
	 cSTA_RUN: 
        THIS^.sta_RUN();
	cSTA_RUNBusy:
        THIS^.sta_RUNBusy();
END_CASE;
END_METHOD

END_FUNCTION_BLOCK

// POUs/Controller/Lvl2/HPS (Heat Press Shirt Station)/FB_DtChnToLine_ChargeDone
FUNCTION_BLOCK FB_DtChnToLine_ChargeDone
VAR_INPUT
	bolResetError: BOOL;
	pSIf: POINTER TO T_Ctrl_SIf_HPS;
END_VAR
VAR_OUTPUT
	///Error value
	intError: INT;
END_VAR
VAR
	/// Internal Variable
	intStatemachine: INT;
	/// Data not correct
	bolDataBad: BOOL;
	/// Retry Counts for error message
	intCountRetry: INT;
	/// Buffer for Senddata
	aBuffer: ARRAY[0..cDtChnBuffer] OF T_ChargeDone_DtChn;
	/// Pointer for new Input
	intPBufferInput: INT;
	/// Pointer for readout
	intPBufferOutput: INT;
	/// Data Channel Specific Variable
	intIndexOldest: INT;
	/// Date and time of the oldes imput
	dtOldestTag: DT;
	fbGetSystemTime: GETSYSTEMTIME;
	stfileTime: T_FILETIME;
	dtActualTime: DT;
END_VAR
VAR CONSTANT
	cDtChnBuffer: INT := 20;
	cSTA_SUB_Data_Init: INT := 900;
	cSTA_SUB_Data_WaitForJob: INT := 902;
	cSTA_SUB_Data_SendData: INT := 904;
	cSTA_SUB_Data_Acknowledge: INT := 906;
	cSTA_SUB_Data_Retry: INT := 908;
	cSTA_SUB_Data_Error: INT := 910;
	cDataState_DONE: INT := -1;
	cDataState_Ready: INT := 1;
	cDataState_Retry: INT := -99;
	cDataState_Error: INT := -100;
	cMAX_RETRY: INT := 10;
	/// Error Codes
	cERR_BufferFull: INT := -99;
	cERR_NoSIF: INT := -100;
END_VAR

(*__________________________________________________________________________________________________
¦	
¦	Vistaprint Schweiz GmbH
¦	CH - 8401 Winterthur
¦
¦	www.vistaprint.ch - info@vistaprint.ch
¦___________________________________________________________________________________________________

Function desription:
Datachannel to send data to Lince Controller
Insert new Job with Method Creat in a Buffer
Send buffer elements if Linecontroller is ready


History:
Version		Date			Author		Comment
---------------------------------------------------------------------------------------------------
0.00.1		26.08.2013		AVM/PRE		Start history


___________________________________________________________________________________________________*)

// Data Channel to Receive Data from Line Controller
// Startup check States
IF (pSIf <> 0) THEN
	IF (intStatemachine < cSTA_SUB_Data_Init) THEN
		intStatemachine := cSTA_SUB_Data_Init;
	END_IF
ELSE
	intError := cERR_NoSIF;
END_IF

CASE intStatemachine OF
	cSTA_SUB_Data_Init:
		IF pSIf^.DtChnToLine.stChargeDone.intDataState = cDataState_DONE THEN
			intStatemachine := cSTA_SUB_Data_WaitForJob;
		END_IF
		
	cSTA_SUB_Data_WaitForJob:
		// New data arrived
		IF intPBufferInput <> intPBufferOutput THEN
			IF pSIf^.DtChnToLine.stChargeDone.intDataState = cDataState_DONE THEN
				intStatemachine := cSTA_SUB_Data_SendData;
			END_IF
		END_IF
	
	cSTA_SUB_Data_SendData:	
		pSIf^.DtChnToLine.stChargeDone.intLine := aBuffer[intPBufferOutput].intLine;
		pSIf^.DtChnToLine.stChargeDone.dtTimestamp := aBuffer[intPBufferOutput].dtTimestamp;
		pSIf^.DtChnToLine.stChargeDone.intDataState := cDataState_Ready;
		intStatemachine := cSTA_SUB_Data_Acknowledge;	
		
	cSTA_SUB_Data_Acknowledge:	
		IF pSIf^.DtChnToLine.stChargeDone.intDataState = cDataState_DONE THEN
			// Data read from Line Controller
			// Reset Buffer Element
			aBuffer[intPBufferOutput].dtTimestamp := DINT_TO_DT(0);
			aBuffer[intPBufferOutput].intDataState := 0;
			aBuffer[intPBufferOutput].intLine := 0;
			// Increase Read out pointer
			IF intPBufferOutput < cDtChnBuffer THEN
				intPBufferOutput := intPBufferOutput + 1;
			ELSE
				intPBufferOutput := 0;
			END_IF
			intStatemachine := cSTA_SUB_Data_WaitForJob;
			
		ELSIF pSIf^.DtChnToLine.stChargeDone.intDataState = cDataState_Retry THEN
			intStatemachine := cSTA_SUB_Data_Retry;
		ELSIF pSIf^.DtChnToLine.stChargeDone.intDataState = cDataState_Error THEN
			intStatemachine := cSTA_SUB_Data_Error;
		END_IF
		
	cSTA_SUB_Data_Retry:
			IF intCountRetry < cMAX_RETRY THEN
				intCountRetry := intCountRetry + 1;
				intStatemachine := cSTA_SUB_Data_SendData;
			ELSE
				intStatemachine := cSTA_SUB_Data_Error;
			END_IF

	cSTA_SUB_Data_Error:
		intError := intCountRetry;
		IF bolResetError = TRUE THEN
			intStatemachine := cSTA_SUB_Data_WaitForJob;
		END_IF
			
END_CASE

METHOD Creat : INT
VAR_INPUT
	In_intLine: INT;
END_VAR
// Insert a new Job to send at Line controller
// Only insert the job, if the buffer is not full, next input dosn't cross input and Outputpointer

// Get Systemtime
fbGetSystemTime(timeLoDW=>stfileTime.dwLowDateTime, timeHiDW=>stfileTime.dwHighDateTime);
dtActualTime := FILETIME_TO_DT( stfileTime );

IF ((intPBufferInput + 1) = intPBufferOutput) OR ((intPBufferInput = cDtChnBuffer) AND (intPBufferOutput = 0)) THEN
	Creat := cERR_BufferFull;
ELSE
	aBuffer[intPBufferInput].intLine := In_intLine;
	aBuffer[intPBufferInput].dtTimestamp := dtActualTime;
	IF intPBufferInput < cDtChnBuffer THEN
		intPBufferInput := intPBufferInput + 1;
	ELSE
		intPBufferInput := 0;
	END_IF
	Creat := intPBufferInput;
END_IF
END_METHOD

END_FUNCTION_BLOCK

// POUs/Controller/Lvl2/HPS (Heat Press Shirt Station)/FB_HPS
FUNCTION_BLOCK FB_HPS EXTENDS FB_CtrlBase
VAR_INPUT
	/// Sensor Counter into the system
	In_bolCounterIn1: BOOL;
	In_bolCounterIn2: BOOL;
	/// Sensor Counter out of the system
	In_bolCounterOut1: BOOL;
	In_bolCounterOut2: BOOL;
	/// Signal to bring a T-Shirt directly (Line 1 without turning)
	In_bolBringShirtStraight: BOOL;
	/// Signal to bring a T-Shirt turned (Line 2 with hanger rotation unit)
	In_bolBringShirtTurned: BOOL;
	///pointer to function blocks Mergers
	p_fbSLB_S: POINTER TO FB_SLB;
	/// Slide buffer for turned T-Shirts
	p_fbSLB_T: POINTER TO FB_SLB;
	p_fbHRU: POINTER TO FB_HRU;
	p_fbSEP: POINTER TO FB_STB;
END_VAR
VAR_OUTPUT
	/// Interface to HeatPress without LineControl
	Out_ShirtStraightReady: BOOL;
	/// Shirt in SEP6 detected
	Out_ShirtTurnReady: BOOL;
END_VAR
VAR
	/// Specific interface struct for public access
	SIf: T_Ctrl_SIf_HPS;
	/// Interface to Childs
	pSLB_S_CIF: POINTER TO T_Ctrl_CIf;
	pSLB_T_CIF: POINTER TO T_Ctrl_CIf;
	pHRU_CIF: POINTER TO T_Ctrl_CIf;
	pSLB_S_SIF: POINTER TO T_Ctrl_SIf_SLB;
	pSLB_T_SIF: POINTER TO T_Ctrl_SIf_SLB;
	pHRU_SIF: POINTER TO T_Ctrl_SIf_HRU;
	pSLB_WORK_CIF: POINTER TO T_Ctrl_CIf;
	pSEP_CIF: POINTER TO T_Ctrl_CIf;
	pSEP_SIF: POINTER TO T_Ctrl_SIf_STB;
	/// Childs of Drives
	/// List of pointers to Childs
	a_pMultiChildCtrl: ARRAY[0..Base_Const.cMaxNrOfChilds] OF POINTER TO FB_DRV;
	/// List of childs common interface
	a_pMultiChildCIF: ARRAY[0..Base_Const.cMaxNrOfChilds] OF POINTER TO T_Ctrl_CIf;
	/// List of childs specific interface for additional parameters or cur
	a_pMultiChildSIF: ARRAY[0..Base_Const.cMaxNrOfChilds] OF POINTER TO T_Ctrl_SIf_DRV;
	usiNumOfMultiChild: USINT;
	usiNumOfValidPointerMultiChild: USINT;
	/// Function specific variables
	/// Rising Edge detection of Hanger Counter input
	bolRECounterIn1: BOOL;
	bolRECounterIn2: BOOL;
	/// Rising Edge detection of Hanger Counter output
	bolRECounterOut1: BOOL;
	bolRECounterOut2: BOOL;
	/// Loopvariable
	intI: INT;
	/// Index of Drive
	intDriveIndex: INT;
	/// Actual Line to charging
	usiLineAct: USINT;
	/// Charge Job
	aTblCharge: ARRAY[0..cintMaxCharge] OF INT;
	/// Datachannel
	/// Internal Variable Data Channel Variables
	intStatemachine: INT;
	/// Data not correct
	bolDataBad: BOOL;
	/// Data found
	bolDataFound: BOOL;
	/// Retry Counts for error message
	intCountRetry: INT;
	/// Datachannel to send done job
	fbDtChnToLine_ChargeDone: FB_DtChnToLine_ChargeDone;
	intDtChnToLineState: INT;
	/// Var. used for sub sequence refill
	intIndexRefill: INT;
	SubStateMachineRefill: INT;
	udiTimeInStateRefill_ms: UDINT;
	/// Rising Edge detection of SIf.In.bolBringShirtStraight.intern
	bolREBringShirtStraight: BOOL;
	/// Rising Edge detection of SIf.In.bolBringShirtTurned.intern
	bolREBringShirtTurned: BOOL;
	// ADS value changed detection for front shirt request 
	udiRequestFrontShirtOld: UDINT;
	// ADS value changed detection for back shirt request 
	udiRequestBackShirtOld: UDINT;
END_VAR
VAR CONSTANT
	///sub States for RELEASE Function
	cSTA_SUB_INITIALIZED: INT := 500;
	cSTA_SUB_START_ELEMENTS: INT := 502;
	cSTA_SUB_START_CYCLE: INT := 504;
	cSTA_SUB_START_WAIT_CYCLE: INT := 506;
	cSTA_SUB_START_INLET: INT := 510;
	cSTA_SUB_START_FINAL: INT := 511;
	cSTA_SUB_STOP_INLET: INT := 512;
	cSTA_SUB_STOP_ELEMENTS: INT := 516;
	cSTA_SUB_STOP_CYCLE: INT := 518;
	cSTA_SUB_STOP_WAIT_CYCLE: INT := 520;
	cSTA_SUB_STOP_OUTLET: INT := 522;
	cSTA_SUB_STOP_FINAL: INT := 524;
	cSTA_SUB_RUN_WAIT_JOB: INT := 530;
	cSTA_SUB_RUN_SET_PAR: INT := 532;
	cSTA_SUB_RUN_SET_CMD: INT := 534;
	cSTA_SUB_RUN_WAIT_DONE: INT := 536;
	cSTA_SUB_RUN_SET_RELEASE: INT := 538;	// Step for SEP
	cSTA_SUB_RUN_WAIT_RELEASED: INT := 540;	// Step for SEP
	cSTA_SUB_RUN_UPDATE: INT := 542;
	cSTA_SUB_ERROR: INT := 598;
	cSTA_SUB_FINISHED: INT := 600;
END_VAR

(*__________________________________________________________________________________________________
¦	
¦	Vistaprint Schweiz GmbH
¦	CH - 8401 Winterthur
¦
¦	www.vistaprint.ch - info@vistaprint.ch
¦___________________________________________________________________________________________________

Function desription:
Heat Press Shirt Station
This controller brings T-Shirts separated to the Heat press over 2 Slides, 
one is directly, the other ower a Hanger rotation Unit to print the backside of the Shirt
Signal to bring the shirt is over digital Input or Data channel


History:
Version		Date			Author		Comment
---------------------------------------------------------------------------------------------------
0.00.1		12.09.2013		AVM/PRE		Start history
0.00.2		19.09.2013		AVME/PRE	Implement new Base Concept
0.00.3		24.09.2013		AVME/MRU	Changes in sta_RUN in SUB-States cSTA_SUB_RUN_WAIT_DONE / 
										cSTA_SUB_RUN_SET_CMD for Hanger Rotation Unit
										Error 'Excepted Hanger not in Rotation Unit' added
										Sensor Counter out of the system 2 added
0.00.4		03.10.2013		AVME/MRU	New Sensor SEP Hanger Detected added
										T_Ctrl_SIf_HPS_Out for Heatpress without LineControl added
										and calculated in RUN
0.00.5		11.12.2013		AVME/MRU	Add Methode checkChildAlmClass for Error Stop of childs
0.00.6		24.01.2014		AVME/MRU	Add SEP_7b
0.00.7		11.02.2014		AVME/DSC	Inserted ADS channel for shirt request send from heatpress
___________________________________________________________________________________________________*)


IF (me.bolActivate) AND (p_fbSLB_S<>0) AND (p_fbSLB_T<>0) AND (p_fbHRU<>0) AND (THIS^.checkChildPointer()) THEN // cyclic call enabled
	IF (CIf.Info.bolInitDone=FALSE) THEN // first cycle -> init
		CtrlInit();
		CIf.Info.bolInitDone := TRUE;
	ELSE
		CycleStartDuty();
	
		Always();
		
		StateMachine();
		
		CycleEndDuty();
	END_IF
END_IF;

METHOD AddDrive
VAR_INPUT
	p_MultiChild: POINTER TO FB_DRV;
END_VAR

// Method add the pointer address of the buffer zone child controller to the array list.
IF (usiNumOfMultiChild <= (Base_Const.cMaxNrOfChilds-1)) THEN
	// Add buffer zone child controller to list
	a_pMultiChildCtrl[usiNumOfMultiChild] := p_MultiChild;
	// Inc. number of buffer zones
	usiNumOfMultiChild:= usiNumOfMultiChild+1;
	// Check if the pointer is valid
	IF (p_MultiChild<>0) THEN
		usiNumOfValidPointerMultiChild:= usiNumOfValidPointerMultiChild+1;
	END_IF
END_IF
END_METHOD

METHOD PROTECTED Always : BOOL
IF (me.bolChangeBackToAUTO=TRUE) THEN // switch mode to automatic switch off controller
	//me.StateMachine.intStateNext := cSTA_OFFBusy;
	//me.bolChangeBackToAUTO := FALSE; // for cylinder no change to off when switch to automatic!!
END_IF

SUPER^.Always();

// ---------------------------------------------------------------------------------
// check child me and set parent alarm class
checkChildAlmClass();

// ----------------------------------------------------------------------------------
// cyclic actions outside of statemachine

// Count Hangers in Controller
// Hanger In
IF SIf.In.bolCounterIn1.intern = TRUE AND bolRECounterIn1 = FALSE THEN
	bolRECounterIn1 := TRUE;
	SIf.Cur.dinCurrentItemCount := SIf.Cur.dinCurrentItemCount + 1;
ELSIF SIf.In.bolCounterIn1.intern = FALSE THEN
	bolRECounterIn1 := FALSE;
END_IF
IF SIf.In.bolCounterIn2.intern = TRUE AND bolRECounterIn2 = FALSE THEN
	bolRECounterIn2 := TRUE;
	SIf.Cur.dinCurrentItemCount := SIf.Cur.dinCurrentItemCount + 1;
ELSIF SIf.In.bolCounterIn2.intern = FALSE THEN
	bolRECounterIn2 := FALSE;
END_IF
// Hanger Out
IF SIf.In.bolCounterOut1.intern = TRUE AND bolRECounterOut1 = FALSE THEN
	bolRECounterOut1 := TRUE;
	IF SIf.Cur.dinCurrentItemCount > 0 THEN
		SIf.Cur.dinCurrentItemCount := SIf.Cur.dinCurrentItemCount - 1;
	END_IF
ELSIF SIf.In.bolCounterOut1.intern = FALSE THEN
	bolRECounterOut1 := FALSE;
END_IF
IF SIf.In.bolCounterOut2.intern = TRUE AND bolRECounterOut2 = FALSE THEN
	bolRECounterOut2 := TRUE;
	IF SIf.Cur.dinCurrentItemCount > 0 THEN
		SIf.Cur.dinCurrentItemCount := SIf.Cur.dinCurrentItemCount - 1;
	END_IF
ELSIF SIf.In.bolCounterOut2.intern = FALSE THEN
	bolRECounterOut2 := FALSE;
END_IF

// Get Maximal Value of capacity
SIf.Cur.dinMaxCapacity := SIf.Cfg.dinMaxCapacity + pSLB_S_SIF^.Cur.dinMaxCapacity + pSLB_T_SIF^.Cur.dinMaxCapacity;

// ----------------------------------------------------------------------------------
// Always change actions in Base Library
// ----------------------------------------------------------------------------------
// overrule error always from base -> no EOFF State!! in EOFF go to OFF
IF (me.StateMachine.intStateNext = cSTA_EOFFBusy) THEN
	IF (me.StateMachine.intState=cSTA_OFF) THEN
		me.StateMachine.intStateNext := cSTA_OFF;
	ELSE // stay in OFF
		me.StateMachine.intStateNext := cSTA_OFFBusy;
	END_IF
END_IF

// Conditions Always
IF (((me.Alarm.eActivAlmClass=E_AlmClass.EOFF) OR (me.Alarm.eActivAlmClass=E_AlmClass.OFF) OR (me.intCmd=cCMD_OFF))
		 AND (me.StateMachine.intState<>cSTA_ERROR) AND (me.StateMachine.intState<>cSTA_ERRORQuit) AND
		(me.StateMachine.intState<>cSTA_OFF) AND (me.StateMachine.intState<>cSTA_OFFBusy)) THEN
	// alarm evt EOFF, OFF or cmd off
	me.StateMachine.intStateNext := cSTA_OFFBusy;
END_IF
END_METHOD

METHOD checkChildAlmClass : BOOL
//------------------------------------------------------------------------------------------------------
// check child alarm classes
// set me alarm class active if at least one child has an EOFF
IF CheckAllChildAlmClass(E_AlmClass.EOFF) THEN
	CIf.Job.eMe_ActivAlmClass := E_AlmClass.EOFF;
	me.Alarm.bolfp := TRUE;
ELSIF CheckAllChildAlmClass(E_AlmClass.OFF) THEN
	CIf.Job.eMe_ActivAlmClass := E_AlmClass.OFF;
	me.Alarm.bolfp := TRUE;
ELSIF CheckAllChildAlmClass(E_AlmClass.STOP) THEN  // FB_MER needs alarm class STOP
	CIf.Job.eMe_ActivAlmClass := E_AlmClass.STOP;
	me.Alarm.bolfp := TRUE;
ELSE
	IF (me.Alarm.bolfp) THEN
		CIf.Job.eMe_ActivAlmClass := E_AlmClass.NONE; // no reset necessary
		me.Alarm.bolfp := FALSE;
	END_IF
END_IF

//------------------------------------------------------------------------------------------------------
// set alarm class parent of childs
//------------------------------------------------------------------------------------------------------
// set alarm class parent of childs in the case of a parent EOFF or me=OFF or EOFF
IF (CIf.Job.eParent_ActivAlmClass=E_AlmClass.EOFF) THEN
	SetAllChildAlmClass(CIf.Job.eParent_ActivAlmClass);
ELSIF(CIf.Job.eMe_ActivAlmClass=E_AlmClass.EOFF) OR (CIf.Job.eMe_ActivAlmClass=E_AlmClass.OFF) THEN
	SetAllChildAlmClass(CIf.Job.eMe_ActivAlmClass);
ELSE
	// no important alarm for child active
	SetAllChildAlmClass(E_AlmClass.NONE);
END_IF
END_METHOD

METHOD PROTECTED checkChildPointer : BOOL
IF (usiNumOfMultiChild = usiNumOfValidPointerMultiChild) THEN
	checkChildPointer:= TRUE;
ELSE
	checkChildPointer:= FALSE;
END_IF
END_METHOD

METHOD PROTECTED checkStateAllMultiChild : BOOL
VAR_INPUT
	cSTA: INT;
END_VAR
VAR
	ii: INT;
	usiNumOfCheckedChilds: USINT;
END_VAR
// Method check input state of all zones

//Init
checkStateAllMultiChild:= FALSE;
usiNumOfCheckedChilds:= 0;

// Loop over all childs
FOR ii:=0 TO usiNumOfMultiChild-1 BY 1 DO
	// Check state	
	IF (a_pMultiChildCIF[ii]^.Job.intState = cSTA) THEN
		usiNumOfCheckedChilds:= usiNumOfCheckedChilds+1;
	END_IF

END_FOR

// All states equal the input state
IF (usiNumOfCheckedChilds = usiNumOfMultiChild) THEN
	checkStateAllMultiChild:= TRUE;
END_IF
END_METHOD

METHOD PROTECTED CmdToAllMultiChild
VAR_INPUT
	cCMD: INT;
END_VAR
VAR
	ii: INT;
END_VAR
// Method send input command to all existing multi child controller.
FOR ii:=0 TO usiNumOfMultiChild-1 BY 1 DO	
	a_pMultiChildCIF[ii]^.Job.intACmd:= cCMD;
END_FOR
END_METHOD

METHOD PROTECTED CtrlInit : BOOL
VAR
	ii: INT;
	usiChildIndex: USINT;
END_VAR
SUPER^.CtrlInit();
// Add Childs
pSLB_S_CIf := THIS^.AddChild(p_fbSLB_S^);
pSLB_T_CIf := THIS^.AddChild(p_fbSLB_T^);
pHRU_CIf := THIS^.AddChild(p_fbHRU^);
pSEP_CIF := THIS^.AddChild(p_fbSEP^);

//initialize all multi Child controller.
FOR ii:=0 TO usiNumOfMultiChild-1 BY 1 DO	
	a_pMultiChildCIF[ii] := THIS^.AddChild(a_pMultiChildCtrl[ii]^);
	a_pMultiChildSIF[ii] := a_pMultiChildCtrl[ii]^.getCtrlSIf();		
END_FOR

pSLB_S_SIF := p_fbSLB_S^.getCtrlSIf();
pSLB_T_SIF := p_fbSLB_T^.getCtrlSIf();
pHRU_SIF := p_fbHRU^.getCtrlSIf();
pSEP_SIF := p_fbSEP^.getCtrlSIf();
END_METHOD

METHOD DtChnToPLC_NewCharge : BOOL
VAR
	ii: INT;
END_VAR
VAR CONSTANT
	cSTA_SUB_Data_Init: INT := 900;
	cSTA_SUB_Data_WaitForJob: INT := 902;
	cSTA_SUB_Data_CheckData: INT := 904;
	cSTA_SUB_Data_Acknowledge: INT := 906;
	cSTA_SUB_Data_Retry: INT := 908;
	cSTA_SUB_Data_Error: INT := 910;
	
	cDataState_DONE: INT := -1;
	cDataState_Ready: INT := 1;
	cDataState_Retry: INT := -99;
	cDataState_Error: INT := -100;
	cMAX_RETRY: INT := 10;
END_VAR
// Data Channel to Receive Data from Line Controller
// Startup check States
IF intStatemachine < cSTA_SUB_Data_Init THEN
	intStatemachine := cSTA_SUB_Data_Init;
END_IF

CASE intStatemachine OF
	cSTA_SUB_Data_Init:
		IF CIf.Job.intState > cSTA_PON THEN
			intCountRetry := 0;
			SIf.DtChnToPLC.stNewCharge.intDataState := cDataState_DONE;
			intStatemachine := cSTA_SUB_Data_WaitForJob;
		END_IF
		
	cSTA_SUB_Data_WaitForJob:
		// New data arrived
		IF SIf.DtChnToPLC.stNewCharge.intDataState = cDataState_Ready THEN
			bolDataBad := FALSE;
			intStatemachine := cSTA_SUB_Data_CheckData;
		END_IF
	
	cSTA_SUB_Data_CheckData:	
		// Check Data
		IF SIf.DtChnToPLC.stNewCharge.intLine <= 0 THEN
				bolDataBad := TRUE;
				// Set Alarm: SIf.Alm[5].strText := 'False Job Parameter';
				pfbAlarmCtrl^.setAlarm(CIf.Info.intCtrlId,5,0,ADR(SIf.Alm),E_AlmState.RST,CIf.Job.eMe_ActivAlmClass);					
		END_IF 
		
		CASE SIf.DtChnToPLC.stNewCharge.intJob OF
			/////////////////////////////////////////////////////
			// Insert new desiction item
			/////////////////////////////////////////////////////							
			E_DtChnJob.NEW:
				// Set new charge Job
				bolDataFound := FALSE;
				FOR ii := 0 TO cintMaxCharge DO
					IF aTblCharge[ii] = SIf.DtChnToPLC.stNewCharge.intLine THEN
						// Set Alarm: SIf.Alm[4].strText := 'Line to charge already busy, Job not possible';
						pfbAlarmCtrl^.setAlarm(CIf.Info.intCtrlId,4,ii,ADR(SIf.Alm),E_AlmState.RST,CIf.Job.eMe_ActivAlmClass);
						bolDataBad := TRUE;	
						EXIT;					
					ELSIF aTblCharge[ii] = 0 THEN
						aTblCharge[ii] := SIf.DtChnToPLC.stNewCharge.intLine;
						bolDataFound := TRUE;
						EXIT;
					END_IF
				END_FOR
				
				IF ((bolDataFound = FALSE) AND (bolDataBad = FALSE)) THEN
					// Set Alarm: SIf.Alm[6].strText := 'Hashtable full, no more input possible';
					pfbAlarmCtrl^.setAlarm(CIf.Info.intCtrlId,6,0,ADR(SIf.Alm),E_AlmState.RST,CIf.Job.eMe_ActivAlmClass);
					bolDataBad := TRUE;						
				END_IF

			/////////////////////////////////////////////////////
			// Delete ID
			/////////////////////////////////////////////////////			
			E_DtChnJob.DELETE_ID:
				// Init value
				bolDataFound := FALSE;
				// Check if Line not allready exist
				// Do not delete the active one index 0
				FOR ii := 1 TO cintMaxCharge DO
					IF aTblCharge[ii] = SIf.DtChnToPLC.stNewCharge.intLine THEN
						aTblCharge[ii] := 0;
						bolDataFound := TRUE;					
					END_IF
					IF ((bolDataFound = TRUE) AND (ii < cintMaxCharge)) THEN
						aTblCharge[ii] := aTblCharge[ii+1];
					ELSIF ((bolDataFound = TRUE) AND (ii = cintMaxCharge)) THEN
						aTblCharge[ii] := 0;						
					END_IF
				END_FOR
								
			/////////////////////////////////////////////////////
			// Delete Junction
			/////////////////////////////////////////////////////			
			E_DtChnJob.DELETE_JUNCTION:
				// Init value
				bolDataFound := FALSE;
				// Check if Line not allready exist
				// Do not delete the active one index 0
				FOR ii := 1 TO cintMaxCharge DO
					IF aTblCharge[ii] = SIf.DtChnToPLC.stNewCharge.intLine THEN
						aTblCharge[ii] := 0;
						bolDataFound := TRUE;					
					END_IF
					IF ((bolDataFound = TRUE) AND (ii < cintMaxCharge)) THEN
						aTblCharge[ii] := aTblCharge[ii+1];
					ELSIF ((bolDataFound = TRUE) AND (ii = cintMaxCharge)) THEN
						aTblCharge[ii] := 0;						
					END_IF
				END_FOR

			/////////////////////////////////////////////////////
			// Delete ALL
			/////////////////////////////////////////////////////			
			E_DtChnJob.DELETE_ALL:
				// Check if RF ID not allready exist
				FOR ii := 0 TO cintMaxCharge DO
					aTblCharge[ii] := 0;					
				END_FOR
				intStatemachine := cSTA_SUB_Data_Acknowledge;
		ELSE
			bolDataBad := TRUE;
			// Set Alarm: SIf.Alm[5].strText := 'False Job Parameter';
			pfbAlarmCtrl^.setAlarm(CIf.Info.intCtrlId,5,0,ADR(SIf.Alm),E_AlmState.RST,CIf.Job.eMe_ActivAlmClass);					
		END_CASE

		IF bolDataBad = TRUE THEN
			IF intCountRetry >= cMAX_RETRY THEN
				intStatemachine := cSTA_SUB_Data_Error;
			ELSE
				intCountRetry := intCountRetry + 1;
				intStatemachine := cSTA_SUB_Data_Retry;
			END_IF	
		ELSE
			intStatemachine := cSTA_SUB_Data_Acknowledge;
		END_IF
		
		
	cSTA_SUB_Data_Acknowledge:	
		// Delete all values
		SIf.DtChnToPLC.stNewCharge.intLine := 0;
		SIf.DtChnToPLC.stNewCharge.intJob := 0;
		// Acknowledge communication
		SIf.DtChnToPLC.stNewCharge.intDataState := cDataState_DONE;
		intStatemachine := cSTA_SUB_Data_WaitForJob;
		
	cSTA_SUB_Data_Retry:
		SIf.DtChnToPLC.stNewCharge.intDataState := cDataState_Retry;
		intStatemachine := cSTA_SUB_Data_WaitForJob;

	cSTA_SUB_Data_Error:
		SIf.DtChnToPLC.stNewCharge.intDataState := cDataState_Error;
		// Set Alarm: SIf.Alm[7].strText := 'Data Channel Error Receive Data';
		pfbAlarmCtrl^.setAlarm(CIf.Info.intCtrlId,7,0,ADR(SIf.Alm),E_AlmState.RST,CIf.Job.eMe_ActivAlmClass);										
		IF CIf.Job.bolAlmReset = TRUE THEN
			intStatemachine := cSTA_SUB_Data_Init;
		END_IF
			
END_CASE
END_METHOD

METHOD FB_init : BOOL
VAR_INPUT
	///if TRUE, the retain variables are initialized (warm start / cold start)
	bInitRetains: BOOL;
	///if TRUE, the instance afterwards gets moved into the copy code (online change)
	bInCopyCode: BOOL;
END_VAR
VAR
	udiTaskCnt: UDINT;
	ii: UINT;
END_VAR
//------------------------------------------------------------------------------------------------------------------------
// to manually change in new FUB implementation!!!
// define valid commands for this controller
FOR ii:= 0 TO (SIZEOF(CIf.Job.aCmdList)/SIZEOF(CIf.Job.aCmdList[0])-1) BY 1 DO
	IF (CIf.Job.aCmdList[ii].intCmd=cCMD_INITIALIZED) THEN
		// found first empty array element
		EXIT;
	END_IF
END_FOR
CIf.Job.aCmdList[ii].intCmd := cCMD_RUN;
CIf.Job.aCmdList[ii].strName := 'Run'; 
CIf.Job.aCmdList[ii].bolAvailable := TRUE;
ii := ii +1;
CIf.Job.aCmdList[ii].intCmd := cCMD_STOP;
CIf.Job.aCmdList[ii].strName := 'Stop'; 
CIf.Job.aCmdList[ii].bolAvailable := TRUE;
ii := ii +1;


// set name of class/typ
CIf.Info.strType := 'FB_HPS'; 

// set alarm class
SIf.Alm[1].eAlmClass := E_AlmClass.EOFF;
SIf.Alm[1].strText := 'Communication Error to Line Controller'; 
SIf.Alm[2].eAlmClass := E_AlmClass.EOFF;
SIf.Alm[2].strText := 'Emergency Button pressed';
SIf.Alm[3].eAlmClass := E_AlmClass.INFO;
SIf.Alm[3].strText := 'Communication Error to Line Controller'; 
SIf.Alm[4].eAlmClass := E_AlmClass.INFO;
SIf.Alm[4].strText := 'Line to charge already busy, Job not possible';
SIf.Alm[5].eAlmClass := E_AlmClass.INFO;
SIf.Alm[5].strText := 'False Job Parameter';
SIf.Alm[6].eAlmClass := E_AlmClass.INFO;
SIf.Alm[6].strText := 'Hashtable full, no more input possible';
SIf.Alm[7].eAlmClass := E_AlmClass.INFO;
SIf.Alm[7].strText := 'Data Channel Error Receive Data';
SIf.Alm[8].eAlmClass := E_AlmClass.INFO;
SIf.Alm[8].strText := 'Data Channel Error Send Data';

//*******************************************************************************
// initial values
//*******************************************************************************
// software configuration
CIf.SwCfg.bolExist := TRUE;
CIf.SwCfg.bolSimulation := FALSE;

// Configuration
SIf.Cfg.bolDtChToLine_send := TRUE;

// parmeter
SIf.Par.udiTimeDriveStart_ms := 2000;
SIf.Par.udiTimeDriveStop_ms := 500;
SIf.Par.udiIntervalBufferFilling_ms:= 2000;
END_METHOD

METHOD PROTECTED getCmdState : STRING
VAR_INPUT
	intCmdState: INT;
	bolState: BOOL;
END_VAR
getCmdState := SUPER^.getCmdState(intCmdState:=intCmdState,bolState:=bolState); // get global/base defined cmds/states
IF (getCmdState='') THEN // global not defined get local
	// get string cmd/state string information in runtime
	IF (bolState=FALSE) THEN
		// cmd's
	ELSE
	
	// cmd's
		CASE intCmdState OF
				
			// SUB States
			cSTA_SUB_INITIALIZED:
				getCmdState := 'cSTA_SUB_INITIALIZED';
			cSTA_SUB_START_CYCLE:
				getCmdState := 'cSTA_SUB_START_CYCLE';
			cSTA_SUB_START_Wait_CYCLE:
				getCmdState := 'cSTA_SUB_START_Wait_CYCLE';
			cSTA_SUB_START_ELEMENTS:
				getCmdState := 'cSTA_SUB_START_ELEMENTS';
			cSTA_SUB_START_INLET:
				getCmdState := 'cSTA_SUB_START_INLET';
			cSTA_SUB_START_FINAL:
				getCmdState := 'cSTA_SUB_START_FINAL';
		
			cSTA_SUB_STOP_INLET:
				getCmdState := 'cSTA_SUB_STOP_INLET';
			cSTA_SUB_STOP_CYCLE:
				getCmdState := 'cSTA_SUB_STOP_CYCLE';
			cSTA_SUB_STOP_Wait_CYCLE:
				getCmdState := 'cSTA_SUB_STOP_Wait_CYCLE';
			cSTA_SUB_STOP_ELEMENTS:
				getCmdState := 'cSTA_SUB_STOP_ELEMENTS';
			cSTA_SUB_STOP_OUTLET:
				getCmdState := 'cSTA_SUB_STOPP_OUTLET';
			cSTA_SUB_ERROR:
				getCmdState := 'cSTA_SUB_ERROR';
			cSTA_SUB_FINISHED:
				getCmdState := 'cSTA_SUB_FINISHED';

			cSTA_SUB_RUN_WAIT_JOB:
				getCmdState := 'cSTA_SUB_RUN_WAIT_JOB';
			cSTA_SUB_RUN_SET_PAR:
				getCmdState := 'cSTA_SUB_RUN_SET_PAR';
			cSTA_SUB_RUN_SET_CMD:
				getCmdState := 'cSTA_SUB_RUN_SET_CMD';
			cSTA_SUB_RUN_WAIT_DONE:
				getCmdState := 'cSTA_SUB_RUN_WAIT_DONE';
			cSTA_SUB_RUN_UPDATE:
				getCmdState := 'cSTA_SUB_RUN_UPDATE';

		END_CASE;
	END_IF
END_IF
END_METHOD

METHOD getCtrlSIf : POINTER TO T_Ctrl_SIf_HPS
getCtrlSIf := ADR(SIf);
END_METHOD

METHOD PROTECTED IoInBridge : BOOL
// digitale and analoge inputs read from hardware or forcing
SIf.In.bolCounterIn1.map := THIS^.In_bolCounterIn1;
SIf.In.bolCounterIn2.map := THIS^.In_bolCounterIn2;
SIf.In.bolCounterOut1.map := THIS^.In_bolCounterOut1;
SIf.In.bolCounterOut2.map := THIS^.In_bolCounterOut2;
SIf.In.bolBringShirtStraight .map := THIS^.In_bolBringShirtStraight;
SIf.In.bolBringShirtTurned .map := THIS^.In_bolBringShirtTurned;

IF (CIf.SwCfg.bolSimulation = FALSE) THEN
	getInBol(CIf.Job.bolIoForce,ADR(SIf.In.bolCounterIn1));
	getInBol(CIf.Job.bolIoForce,ADR(SIf.In.bolCounterIn2));
	getInBol(CIf.Job.bolIoForce,ADR(SIf.In.bolCounterOut1));
	getInBol(CIf.Job.bolIoForce,ADR(SIf.In.bolCounterOut2));
	getInBol(CIf.Job.bolIoForce,ADR(SIf.In.bolBringShirtStraight));
	getInBol(CIf.Job.bolIoForce,ADR(SIf.In.bolBringShirtTurned));
ELSE
	//simulation of global IO
END_IF
END_METHOD

METHOD PROTECTED IoOutBridge : BOOL
// digitale and analoge inputs read from hardware or forcing
IF (CIf.SwCfg.bolSimulation = FALSE) THEN
	// check interlocks to prevent damages
	IF (CIf.Job.bolIlkOverwrite=FALSE) THEN
	
		;
	END_IF
	
	// Outputs for Interface to HeatPress without LineControl
	setOutBol(CIf.Job.bolIoForce ,ADR(SIf.Out.bolShirtStraightReady));
	setOutBol(CIf.Job.bolIoForce ,ADR(SIf.Out.bolShirtTurnReady));	
	THIS^.Out_ShirtStraightReady := SIf.Out.bolShirtStraightReady.map;
	THIS^.Out_ShirtTurnReady := SIf.Out.bolShirtTurnReady.map;
	
END_IF
END_METHOD

METHOD RefillTurnedLine
VAR
	/// Loop variable
	ii: INT;
END_VAR
// Simulation
IF (CIf.SwCfg.bolSimulation) THEN
;
END_IF
	
	
// Method refill all zones
CASE SubStateMachineRefill OF		
			
	// Check space in buffer X
	//-------------------------------
	0:
		// Check if number of hangers "per Pulse" have space in the next buffer
		// Condition: (zone[X].NumOfHangers + zone[ X + 1] .NumOfHangersPerPuls) < zone[X].MaxCapacity   			
		IF ((pSEP_SIF^.Cur.dinNumOfHangersInBuffer < pSEP_SIF^.Cfg.dinMaxCapacity) AND 
			(pSLB_T_SIF^.Cur.dinNumOfHangersInBuffer <> 0) AND (pSLB_T_SIF^.Cur.bolHangerDetected = TRUE)) THEN
			
			// Send release command to buffer zone X+1
			pSLB_T_CIF^.Job.intACmd:= SLB_CmdState.cCMD_RELEASE;	
			SubStateMachineRefill:= 1;						
		END_IF
	
	// Check if zone X+1 is released
	//-------------------------------
	1:
		IF(pSLB_T_CIF^.Job.intACmd = BASE_PLC.cCMD_DONE)THEN
			// Send stop command to buffer zone X+1
			SubStateMachineRefill:= 2;
			// Counter correction if no counter at inside of Buffer
			IF pSEP_SIF^.Cfg.bolHasBufferFullSensor = FALSE THEN
				pSEP_SIF^.Cur.dinNumOfHangersInBuffer := pSEP_SIF^.Cur.dinNumOfHangersInBuffer + 1;
			END_IF
		END_IF	
	
	// Check if zone X+1 is stopped
	//-------------------------------
	2:
		udiTimeInStateRefill_ms:= 0;
		SubStateMachineRefill:= 3;
		pHRU_CIF^.Job.intACmd := cCMD_RUN;	// Set Command to HRU				
	
	// Check if HRU is done
	//-------------------------------
	3: 
		IF (pHRU_CIf^.Job.intACmd = cSTA_DONE) THEN							// Hanger Rotation Unit done
			SubStateMachineRefill:= 4;
		END_IF

		
	// Break
	//-------------------------------
	4:	
		// Increment time in state	
		udiTimeInStateRefill_ms:= udiTimeInStateRefill_ms + me.FUBInfo.udiSample_ms;
		IF (udiTimeInStateRefill_ms > SIf.Par.udiIntervalBufferFilling_ms) THEN
			// Back to first state
			SubStateMachineRefill:= 0;	
		END_IF
		
END_CASE
END_METHOD

METHOD PROTECTED sta_OFF : BOOL
// state implemetation
//--------------------------------------------------------------------------------------
// Entry action
	IF (me.StateMachine.intState<>me.StateMachine.intStateLastCycle) THEN
		me.StateMachine.intStateLastCycle := me.StateMachine.intState;
		
	END_IF


//--------------------------------------------------------------------------------------
// Cyclic action
	IF (me.StateMachine.intState=me.StateMachine.intStateLastCycle) THEN
		
		;
		
		
		// State Change Condition
		IF (me.intCmd=cCMD_RUN) THEN
			me.StateMachine.intStateNext :=  cSTA_RUNBusy;
		END_IF
	END_IF




//--------------------------------------------------------------------------------------
// Exit action
	IF (me.StateMachine.intState<>me.StateMachine.intStateNext) THEN
		;
	END_IF
END_METHOD

METHOD PROTECTED sta_RUN : BOOL
// state implemetation
//--------------------------------------------------------------------------------------
// Entry action
	IF (me.StateMachine.intState<>me.StateMachine.intStateLastCycle) THEN
		me.StateMachine.intStateLastCycle := me.StateMachine.intState;
		
		me.SubStateMachine.intState := cSTA_SUB_RUN_WAIT_JOB; // init sub state machine
		me.SubStateMachine.intStateNext := cSTA_SUB_RUN_WAIT_JOB; // init sub state machine

	END_IF


//--------------------------------------------------------------------------------------
// Cyclic action
	IF (me.StateMachine.intState=me.StateMachine.intStateLastCycle) THEN

		// Simulation
		IF (CIf.SwCfg.bolSimulation) THEN
			;
		END_IF

		// Get emptying command from Line with Data Channel
		// Communication to the Line Controll over Data Channel
		THIS^.DtChnToPLC_NewCharge();
		fbDtChnToLine_ChargeDone.bolResetError := CIf.Job.bolAlmReset;
		fbDtChnToLine_ChargeDone.pSIf := ADR(SIf);
		fbDtChnToLine_ChargeDone();
		IF fbDtChnToLine_ChargeDone.intError <> 0 THEN
			// Set Alarm: SIf.Alm[8].strText := 'Data Channel Error Send Data';
			pfbAlarmCtrl^.setAlarm(CIf.Info.intCtrlId,8,fbDtChnToLine_ChargeDone.intError,ADR(SIf.Alm),E_AlmState.RST,CIf.Job.eMe_ActivAlmClass);	
		END_IF
	
		// Start Cycle with substates	
		//--------------------------------------------------------------------------------------
		// sub state machine for sequence
		CASE me.SubStateMachine.intState OF
			//--------------------------------------------------------------------------------------
			
			cSTA_SUB_RUN_WAIT_JOB:
				//--------------------------------------------------------------
				// Job can be set on 3 different ways:
				// 1. Over data channel from Line Controller
				// 2. By digital input (output on heatpress)
				// 3. Over ADS data channel from heatpress
				//--------------------------------------------------------------
				IF ((aTblCharge[0] > 0) 
				OR (SIf.In.bolBringShirtStraight.intern AND NOT bolREBringShirtStraight)
				OR (SIf.In.bolBringShirtTurned.intern AND NOT bolREBringShirtTurned)
				OR (SIf.Ads.stRead.udiRequestBackShirt <> udiRequestBackShirtOld)
				OR (SIf.Ads.stRead.udiRequestFrontShirt <> udiRequestFrontShirtOld)) THEN																	
					me.SubStateMachine.intStateNext := cSTA_SUB_RUN_SET_CMD;
				END_IF
							
				// Interface to HeatPress without LineControl
				SIf.Out.bolShirtStraightReady.intern := pSLB_S_SIF^.Cur.bolHangerDetected; 	// Sensor SEP7 has Hanger detected
				SIf.Out.bolShirtTurnReady.intern := pSEP_SIF^.Cur.bolHangerDetected; // pSLB_T_SIF^.Cur.bolHangerDetected;		// Sensor SEP6 has Hanger detected
				
			cSTA_SUB_RUN_SET_CMD:
				// Digital Input or ADS has priority to the data channel
				// get the correct Common interface to set the RELEASE Command
				IF ((SIf.In.bolBringShirtStraight.intern = TRUE) OR (SIf.Ads.stRead.udiRequestFrontShirt <> udiRequestFrontShirtOld)) THEN
					udiRequestFrontShirtOld:= SIf.Ads.stRead.udiRequestFrontShirt; 
					pSLB_WORK_CIF := pSLB_S_CIF;
				ELSIF ((SIf.In.bolBringShirtTurned.intern = TRUE) OR (SIf.Ads.stRead.udiRequestBackShirt <> udiRequestBackShirtOld)) THEN
					udiRequestBackShirtOld:= SIf.Ads.stRead.udiRequestBackShirt; 
					pSLB_WORK_CIF := pSEP_CIF; //pSLB_T_CIF;	
				ELSIF (aTblCharge[0] = 1) THEN
					// If job from Datachannel, save the line number
					usiLineAct := INT_TO_USINT(aTblCharge[0]);
					pSLB_WORK_CIF := pSLB_S_CIF;
				ELSIF (aTblCharge[0] = 2) THEN
					// If job from Datachannel, save the line number
					usiLineAct := INT_TO_USINT(aTblCharge[0]);
					pSLB_WORK_CIF := pSEP_CIF; //pSLB_T_CIF;
				END_IF
				
